# B&R Automation Studio project ACOPOStrak_DATech_Pilot (part 4)

#### Types.typ - Local data types
```iecst
(*estimate assembly power consumption and distribution*)
(*interface structure*)

TYPE
	TrakDesignType : 	STRUCT
		AssemblyRef : REFERENCE TO McAssemblyType; (*assembly reference - ADR(gAssembly_1)*)
		AssemblyName : STRING[32]; (*assembly name - 'gAssembly_1'*)
		EnableCalc : BOOL; (*enable*)
		CmdReset : BOOL; (*command reset peak values*)
		CmdSaveReport : BOOL; (*command save report to file*)
		CmdRecordToolData : BOOL; (*command activate recording of TrakDesign-Tool data*)
		ParaShuttleType : TrakDesignShuttleTypeEnum; (*parameter shuttle type
SA100_50D......8F1SA.100.xxxxxx-1  50mm double sided magnet
SA102_50N......8F1SA.102.xxxxxx-1  50mm single sided magnet
SA201_100D....8F1SA.201.xxxxxx-1  100mm double sided magnet
SA203_100N....8F1SA.203.xxxxxx-1  100mm single sided magnet
SA104_50DS....8F1SA.104.xxxxxx-1  50mm double sided skewed magnet
SA106_50NS....8F1SA.106.xxxxxx-1  50mm single sided skewed magnet
SB308_210N....8F1SB.308.xxxxxx-1  21magnet pole single sided magnet*)
		ParaTempAmbient : REAL; (*parameter ambient air temperature [°C]*)
		ParaMechShuttleIx : UINT; (*parameter mechanical check - use shuttle index*)
		ParaFileDevice : STRING[32]; (*parameter FileDevice*)
		ParaFileNameReport : STRING[32]; (*parameter report file name - file extention .csv mandatory*)
		ParaFileNameToolData : STRING[32]; (*parameter TrakDesign-Tool data file name - file extention .dat mandatory*)
		ParaFileCsvStyle : USINT; (*parameter file csv style
0..english
1..german
2..mathlab*)
		ParaToolDataPrescale : USINT; (*parameter TrakDesign-Tool data prescaler - record TrakDesign-Tool data every x task cycles*)
		Message : STRING[256]; (*message*)
		TimeAsmPowerOn : REAL; (*monitor time elapsed since AsmPowerOn*)
		TimeShuttlesMoving : REAL; (*monitor time shuttles moving - for stabile Avg values process needs to run for >120sec*)
		TimeReset : REAL; (*monitor time elapsed since CmdReset*)
		TimeRecordToolDataActive : REAL; (*monitor time recording of TrakDesign-Tool data active*)
		NumShuttles : UINT; (*monitor number of shuttles present*)
		Carrier : TrakDesignCarrierType;
		Payload : ARRAY[1..8]OF TrakDesignPayloadType;
		Shuttle : ARRAY[1..TRAK_MAX_SHUTTLE]OF TrakDesignShuttleType;
		Segment : ARRAY[1..TRAK_MAX_SEGMENT]OF TrakDesignSegmentType;
		Cable : ARRAY[1..TRAK_MAX_POWER_CABLE]OF TrakDesignCableType;
		Supply : ARRAY[1..TRAK_MAX_POWER_SUPPLY]OF TrakDesignSupplyType;
		MainSupply : TrakDesignMainSupplyType;
		Mech : TrakDesignMechType;
	END_STRUCT;
	TrakDesignCarrierType : 	STRUCT
		ParaMass : LREAL; (*parameter payload carrier mass [kg]*)
		ParaMassCenterX : LREAL; (*parameter payload carrier mass center of gravity offset X [m] (measured from center of shuttle, sign according to the shuttle coordinate system)*)
		ParaMassCenterY : LREAL; (*parameter payload carrier mass center of gravity offset Y [m] (measured from center of shuttle, sign according to the shuttle coordinate system)*)
		ParaMassCenterZ : LREAL; (*parameter payload carrier mass center of gravity offset Z [m] (measured from center of shuttle, sign according to the shuttle coordinate system)*)
		ParaMassInertiaZZ : LREAL; (*parameter payload carrier inertia ZZ [kgm? (with respect to the center of gravity of the carrier - set to 0.0 if unknown)*)
	END_STRUCT;
	TrakDesignPayloadType : 	STRUCT
		ParaName : STRING[32]; (*parameter payload name (free definable name for identification of payload in report and mathlab)*)
		ParaMass : LREAL; (*parameter payload product mass [kg]*)
		ParaMassCenterX : LREAL; (*parameter payload product mass center of gravity offset X [m] (measured from center of shuttle, sign according to the shuttle coordinate system)*)
		ParaMassCenterY : LREAL; (*parameter payload product mass center of gravity offset Y [m] (measured from center of shuttle, sign according to the shuttle coordinate system)*)
		ParaMassCenterZ : LREAL; (*parameter payload product mass center of gravity offset Z [m] (measured from center of shuttle, sign according to the shuttle coordinate system)*)
		ParaMassInertiaZZ : LREAL; (*parameter payload product inertia ZZ [kgm? (with respect to the center of gravity of the payload - set to 0.0 if unknown)*)
		ParaExtFrictionX : LREAL; (*parameter external process friction [N] (sign according to the shuttle movement direction)*)
		ParaExtFrictionVelX : LREAL; (*parameter external process velocity-friction [N/(m/s)] (sign according to the shuttle movement direction)*)
		ParaExtForceX : LREAL; (*parameter external process force X [N] (sign according to the shuttle coordinate system)*)
		ParaExtForceY : LREAL; (*parameter external process force Y [N] (sign according to the shuttle coordinate system)*)
		ParaExtForceZ : LREAL; (*parameter external process force Z [N] (sign according to the shuttle coordinate system)*)
		ParaExtForceAppPointX : LREAL; (*parameter external process force application point offset X [m] (measured from center of shuttle, sign according to the shuttle coordinate system)*)
		ParaExtForceAppPointY : LREAL; (*parameter external process force application point offset Y [m] (measured from center of shuttle, sign according to the shuttle coordinate system)*)
		ParaExtForceAppPointZ : LREAL; (*parameter external process force application point offset Z [m] (measured from center of shuttle, sign according to the shuttle coordinate system)*)
	END_STRUCT;
	TrakDesignShuttleType : 	STRUCT
		ParaPayloadIx : USINT; (*parameter payload index*)
		ParaAutoPayload : USINT; (*parameter autmatic payload selection 0..set PayloadIx explicit / 1..get payload index from ShSelCtrlParSet index*)
		ParaInitialOrientationFlip : INT; (*the initial orientation is different from the one indicated or located.[-]
  1 --> initial orientation is identical with the indicated or located one
 -1 --> initial orientation is different with the indicated or located one *)
		ID : UINT; (*shuttle ID*)
		Vel : LREAL; (*shuttle velocity [m/s]*)
		Acc : LREAL; (*shuttle acceleration [m/s?*)
		Area : USINT; (*shuttle is in area 0..straight / 1..circular / 2..diverter*)
		Force : REAL; (*shuttle thrust force [N]*)
		Current : REAL; (*shuttle current [A]*)
		PowerCalcAct : REAL; (*monitor current shuttle power [W]*)
		PowerCalcAvg : REAL; (*monitor filtered shuttle power [W]*)
		VelStraightPeak : REAL; (*report peak shuttle velocity in straight trak area [m/s]*)
		AccStraightPeak : REAL; (*report peak shuttle acceleration in straight trak area [m/s?*)
		VelCircularPeak : REAL; (*report peak shuttle velocity in circular trak area [m/s]*)
		AccCircularPeak : REAL; (*report peak shuttle acceleration in circular trak area [m/s?*)
		VelDiverterPeak : REAL; (*report peak shuttle velocity in diverter area [m/s]*)
		AccDiverterPeak : REAL; (*report peak shuttle acceleration in diverter area [m/s?*)
		ForcePeak : REAL; (*report peak shuttle thrust Force [N]*)
		CurrentPeak : REAL; (*report peak shuttle current [A]*)
		PowerCalcActPeak : REAL; (*report peak current shuttle power [W]*)
		PowerCalcAvgPeak : REAL; (*report peak filitered shuttle power [W]*)
		CoilDisabled : USINT; (*report reduced force due to temporary disabled stator coil*)
	END_STRUCT;
	TrakDesignSegmentType : 	STRUCT
		ParaName : STRING[32]; (*parameter segment name
name of segment reference variable of type McSegmentType connected to this segment in SystemDesigner*)
		ParaType : TrakDesignSegmentTypeEnum; (*parameter segment type
TYPE_AA
TYPE_AB
TYPE_BA
TYPE_BB*)
		ParaIxCable : USINT; (*parameter segment connected to cable index*)
		ID : UINT; (*segment ID*)
		PowerCalcAct : REAL; (*monitor current segment power [W]*)
		PowerCalcAvg : REAL; (*monitor filtered segment power [W]*)
		PowerCalcActPeak : REAL; (*report peak current segment power [W]*)
		PowerCalcAvgPeak : REAL; (*report peak filtered segment power [W]*)
		PowerCalcLoss : REAL; (*monitor current segment loss [W]*)
		PowerCalcLoad : REAL; (*monitor filtered segment Load [W]*)
		PowerCalcLossPeak : REAL; (*report peak current segment loss [W]*)
		PowerCalcLoadPeak : REAL; (*report peak filtered segment Load [W]*)
		CurrentBalancer : REAL; (*monitor balancer current [A]*)
		CurrentBalancerPeak : REAL; (*report peak balancer current [A]*)
		CoilDisabled : USINT; (*report reduced force due to temporary disabled stator coil*)
	END_STRUCT;
	TrakDesignCableType : 	STRUCT
		ParaLength : REAL; (*parameter cable length [m]*)
		ParaIxSupply : USINT; (*parameter cable connected to PowerSupply index*)
		PowerCalcAct : REAL; (*monitor current cable power [W]*)
		PowerCalcAvg : REAL; (*monitor filtered cable power [W]*)
		PowerCalcActPeak : REAL; (*report peak cable shuttle power [W]*)
		PowerCalcAvgPeak : REAL; (*report peak cable shuttle power [W]*)
		VoltageDropAct : REAL; (*monitor voltage drop [V]*)
		VoltageDropActPeak : REAL; (*report peak voltage drop [V]*)
	END_STRUCT;
	TrakDesignSupplyType : 	STRUCT
		ParaName : STRING[32]; (*parameter supply name
name of supply reference variable of type McAxisType connected to this BC032 in SystemDesigner*)
		ParaType : TrakDesignSupplyTypeEnum; (*parameter supply type
PS080...80PS080X3.10-01         1kW standalone power supply (ACOPOSmicro)
BC032...8B0C0320HW00.B00-1 2kW backplane power supply (ACOPOSmulti)*)
		ParaIxSupplyParallel : USINT; (*Parameter supply is parallel connected to supply index / 0..no parallel connection*)
		PowerCalcAct : REAL; (*monitor current supply power [W]*)
		PowerCalcAvg : REAL; (*monitor filtered supply power [W]*)
		PowerCalcActPeak : REAL; (*report peak current supply power [W]*)
		PowerCalcAvgPeak : REAL; (*report peak filitered supply power [W]*)
		PowerCalcRetPeak : REAL; (*report peak current return power [W]*)
		PowerMeasAct : REAL; (*monitor current supply power [W] (measured via IO)*)
		PowerMeasAvg : REAL; (*monitor filtered supply power [W] (measured via IO)*)
		PowerMeasActPeak : REAL; (*report peak current supply power [W] (measured via IO)*)
		PowerMeasAvgPeak : REAL; (*report peak filitered supply power [W] (measured via IO)*)
		PowerMeasRetPeak : REAL; (*report peak current return power [W] (measured via IO)*)
		IoPS080 : TrakDesignSupplyIoPS080Type;
		IoBC032 : TrakDesignSupplyIoBC032Type;
	END_STRUCT;
	TrakDesignSupplyIoPS080Type : 	STRUCT
		ModuleOk : BOOL; (*PS080 IO*)
		CurrentLimitActive : BOOL; (*PS080 IO*)
		Voltage : SINT; (*PS080 IO [V]*)
		Current : INT; (*PS080 IO [0.1A]*)
		CmdClearError : BOOL; (*PS080 IO*)
		ErrorOutput : BOOL; (*PS080 IO*)
		ErrorOverload : BOOL; (*PS080 IO*)
		ErrorPhaseDetection : BOOL; (*PS080 IO*)
		ErrorOvertemperature : BOOL; (*PS080 IO*)
		ErrorOvervoltage : BOOL; (*PS080 IO*)
		ChopperActive : BOOL; (*PS080 IO*)
		ErrorChopperTemperature : BOOL; (*PS080 IO*)
		ErrorBleederTemperature : BOOL; (*PS080 IO*)
		ErrorOutput24VDC : BOOL; (*PS080 IO*)
	END_STRUCT;
	TrakDesignSupplyIoBC032Type : 	STRUCT
		ModuleOk : BOOL; (*8B0C0320 IO module OK*)
		Iout : REAL; (*8B0C0320 IO Actual Output current [A]*)
		Uout : REAL; (*8B0C0320 IO Actual Output voltage [V]*)
		CrOk : BOOL; (*8B0C0320 IO state charging relais 1..OK*)
		StatusRunMode : USINT; (*8B0C0320 IO Operating mode 0..INIT / 1..READY / 2..ACTIVE / 3..ERROR*)
		ErrorsPacked : UDINT; (*8B0C0320 IO ErrorsPacked - Register ERROR_REG*)
		WarningsPacked : UDINT; (*8B0C0320 IO WarningsPacked - Register WARN_REG*)
	END_STRUCT;
	TrakDesignMainSupplyType : 	STRUCT
		PowerCalcAct : REAL; (*monitor current main supply power [W]*)
		PowerCalcAvg : REAL; (*monitor filtered main supply power [W]*)
		PowerCalcActPeak : REAL; (*report peak current main supply power [W]*)
		PowerCalcAvgPeak : REAL; (*report peak filitered main supply power [W]*)
		PowerCalcRetPeak : REAL; (*report peak current main return power [W]*)
		PowerMeasAct : REAL; (*monitor current main supply power [W] (measured via IO)*)
		PowerMeasAvg : REAL; (*monitor filtered main supply power [W] (measured via IO)*)
		PowerMeasActPeak : REAL; (*report peak current main supply power [W] (measured via IO)*)
		PowerMeasAvgPeak : REAL; (*report peak filitered main supply power [W] (measured via IO)*)
		PowerMeasRetPeak : REAL; (*report peak current main return power [W] (measured via IO)*)
	END_STRUCT;
	TrakDesignMechType : 	STRUCT
		ShuttleIx : UINT;
		ShuttleID : UINT;
		PayloadIx : USINT; (*parameter payload index*)
		ResultThrust : BOOL; (*report thrust force 0..ok / 1..force insufficient*)
		ResultMech : BOOL; (*report mechanical failure 0..ok / 1..shuttle leaving guiding rails*)
		GlobalFrame : McFrameType;
		SectorName : STRING[32];
		SectorPosition : LREAL;
		SectorVelocity : LREAL;
		SectorAcceleration : LREAL;
		SectorOrientation : McDirectionEnum;
		SegmentValid : ARRAY[0..3]OF BOOL;
		SegmentID : ARRAY[0..3]OF UINT;
		SegmentName : ARRAY[0..3]OF STRING[32];
		SegmentTyp : ARRAY[0..3]OF TrakDesignSegmentTypeEnum;
		SegmentLength : ARRAY[0..3]OF LREAL;
		SegmentPosition : ARRAY[0..3]OF LREAL;
		SegmentFieldMode : ARRAY[0..3]OF McAcpTrakFieldModeEnum;
	END_STRUCT;
END_TYPE

(*interface TrakDesign shuttle online interaction*)

TYPE
	TrakDesignOnlineFunctionJobType : 	STRUCT
		LockNew : UDINT;
		Axis : McAxisType;
		ShuttleID : UINT;
		Cmd : USINT;
		PayloadIx : USINT;
		spare : ARRAY[0..3]OF UDINT;
		LockEnd : UDINT;
	END_STRUCT;
END_TYPE

(*TrakDesign-Tool data (diagnosis-data)*)

TYPE
	TrakDesignDiagParaType : 	STRUCT
		VersionDataStruct : UDINT := 2;
		VersionMappMotion : ARRAY[0..9]OF USINT;
		VersionTrakDesignTask : ARRAY[0..9]OF USINT;
		CycleTime : REAL;
		Prescaler : USINT;
		ShuttleType : UINT;
		TempAmbient : REAL;
		PayloadCnt : UINT;
		Carrier : TrakDesignDiagParaCarrierType;
		Payload : ARRAY[1..8]OF TrakDesignDiagParaPayloadType;
		SegmentCnt : UINT;
		Segment : ARRAY[1..TRAK_MAX_SEGMENT]OF TrakDesignDiagParaSegmentType;
		CableCnt : UINT;
		Cable : ARRAY[1..TRAK_MAX_POWER_CABLE]OF TrakDesignDiagParaCableType;
		SupplyCnt : UINT;
		Supply : ARRAY[1..TRAK_MAX_POWER_SUPPLY]OF TrakDesignDiagParaSupplyType;
	END_STRUCT;
	TrakDesignDiagParaCarrierType : 	STRUCT
		Mass : LREAL;
		MassCenterX : LREAL;
		MassCenterY : LREAL;
		MassCenterZ : LREAL;
		MassInertiaZZ : LREAL;
	END_STRUCT;
	TrakDesignDiagParaPayloadType : 	STRUCT
		Name : STRING[32];
		Mass : LREAL;
		MassCenterX : LREAL;
		MassCenterY : LREAL;
		MassCenterZ : LREAL;
		MassInertiaZZ : LREAL;
		ExtFrictionX : LREAL;
		ExtFrictionVelX : LREAL;
		ExtForceX : LREAL;
		ExtForceY : LREAL;
		ExtForceZ : LREAL;
		ExtForceAppPointX : LREAL;
		ExtForceAppPointY : LREAL;
		ExtForceAppPointZ : LREAL;
	END_STRUCT;
	TrakDesignDiagParaSegmentType : 	STRUCT
		Ix : UINT;
		ID : UINT;
		Name : STRING[32];
		Type : TrakDesignSegmentTypeEnum;
		IxCable : UINT;
	END_STRUCT;
	TrakDesignDiagParaCableType : 	STRUCT
		Ix : UINT;
		Length : REAL;
		IxSupply : UINT;
	END_STRUCT;
	TrakDesignDiagParaSupplyType : 	STRUCT
		Ix : UINT;
		Type : TrakDesignSupplyTypeEnum;
		IxSupplyParallel : UINT;
	END_STRUCT;
	TrakDesignDiagType : 	STRUCT
		RecordIndex : UDINT;
		Time : REAL;
		MechShuttleIx : UINT;
		MechResultThrust : BOOL;
		MechResultMech : BOOL;
		AddData : ARRAY[0..4]OF LREAL;
		SegmentCnt : UINT;
		Segment : ARRAY[1..TRAK_MAX_SEGMENT]OF TrakDesignDiagSegmentType;
		ShuttleCnt : UINT;
		Shuttle : ARRAY[1..TRAK_MAX_SHUTTLE]OF TrakDesignDiagShuttleType;
	END_STRUCT;
	TrakDesignDiagSegmentType : 	STRUCT
		CalcPower : REAL;
		CalcLoss : REAL;
	END_STRUCT;
	TrakDesignDiagShuttleType : 	STRUCT
		ID : UINT;
		GlobalFrame : McFrameType;
		SectorVelocity : LREAL;
		SectorAcceleration : LREAL;
		SectorOrientation : McDirectionEnum;
		PayloadIx : UINT;
		GripperCnt : UINT;
		GripperSegValid : ARRAY[0..3]OF BOOL;
		GripperSegIx : ARRAY[0..3]OF UINT;
		GripperSegPosition : ARRAY[0..3]OF LREAL;
		GripperSegFieldMode : ARRAY[0..3]OF McAcpTrakFieldModeEnum;
	END_STRUCT;
END_TYPE

(*supply-data (ServoSoft-import-data)*)

TYPE
	TrakDesignSupplyDataType : 	STRUCT
		Time : LREAL;
		Power : ARRAY[0..TRAK_MAX_POWER_SUPPLY]OF REAL;
	END_STRUCT;
END_TYPE

(*enum*)

TYPE
	TrakDesignShuttleTypeEnum :
		(
		SHUTTLE_UNDEFINED := 0,
		SA100_50D := 100, (*8F1SA.100.xxxxxx-1  50mm double sided magnet*)
		SA102_50N := 102, (*8F1SA.102.xxxxxx-1  50mm single sided magnet*)
		SA201_100D := 201, (*8F1SA.201.xxxxxx-1  100mm double sided magnet*)
		SA203_100N := 203, (*8F1SA.203.xxxxxx-1  100mm single sided magnet*)
		SA104_50DS := 104, (*8F1SA.104.xxxxxx-1  50mm double sided skewed magnet*)
		SA106_50NS := 106, (*8F1SA.106.xxxxxx-1  50mm single sided skewed magnet*)
		SHUTTLE_205 := 205, (*internal*)
		SHUTTLE_207 := 207, (*internal*)
		SB308_210N := 1308, (*8F1SB.308.xxxxxx-1  21magnet pole single sided magnet*)
		SHUTTLE_9100 := 9100, (*internal*)
		SHUTTLE_65535 := 65535 (*internal*)
		);
	TrakDesignSegmentTypeEnum :
		(
		SEGMENT_UNDEFINED := 0,
		TYPE_AA := 1, (*AA Straight segment*)
		TYPE_AB := 2, (*AB Curved segment*)
		TYPE_BA := 3, (*BA Curved segment*)
		TYPE_BB := 4 (*BB Circular arc segment*)
		);
	TrakDesignSupplyTypeEnum :
		(
		SUPPLY_UNDEFINED := 0,
		PS080 := 1, (*80PS080X3.10-01 1kW standalone power supply (ACOPOSmicro)*)
		BC032 := 2 (*8B0C0320HW00.B00-1 2kW backplane power supply (ACOPOSmulti)*)
		);
	TrakDesignStepGetShuttleEnum :
		(
		TRAK_DISABLED := 0,
		TRAK_WAIT,
		TRAK_GET_SHUTTLE_INIT,
		TRAK_GET_SHUTTLE,
		TRAK_GET_SHUTTLE_WAIT,
		TRAK_INIT,
		TRAK_READY,
		TRAK_ERROR
		);
END_TYPE
```

#### Variables.var - Local variables
```iecst
(*task interface structure*)
VAR
	TrakDesign : TrakDesignType;
END_VAR
(*online interface*)
VAR
	OnlineFunctionJob : ARRAY[0..19] OF TrakDesignOnlineFunctionJobType;
	ShuttleIxFound : UDINT := 0;
	ShuttleIxAdd : UDINT := 0;
END_VAR
(*general*)
VAR
	RTInfo_0 : RTInfo;
	TCCycleTime : LREAL;
	i : UDINT;
	k : UINT;
	m : UINT;
	ErrorMessage : USINT := 0;
	VersionMcAcpTrak : MoVerStruc_typ := (0);
	VersionTrakDesignTask : MoVerStruc_typ := (0);
END_VAR
(*get shuttle axis*)
VAR
	MC_BR_AsmReadInfo_AcpTrak_0 : MC_BR_AsmReadInfo_AcpTrak;
	MC_BR_AsmGetShuttle_AcpTrak_0 : MC_BR_AsmGetShuttle_AcpTrak;
	StepGetShuttle : TrakDesignStepGetShuttleEnum;
	CyclesWaitGetShuttle : UINT := TRAK_MAX_SHUTTLE * 5;
	CntWait : UINT;
	CntShuttle : UINT;
	CntShuttleIdentPowerOn : UDINT;
	CntShuttleAddedOnline : UDINT;
	CntShuttleDeletedOnline : UDINT;
	ShuttleAxis : ARRAY[1..TRAK_MAX_SHUTTLE] OF McAxisType;
	AssemblyOrientation : REAL := 0.0;
END_VAR
(*shutte & segment power*)
VAR
	MC_BR_ShReadInfo_AcpTrak_0 : ARRAY[1..TRAK_MAX_SHUTTLE] OF MC_BR_ShReadInfo_AcpTrak;
	MC_BR_ShReadSegmentInfo_0 : ARRAY[1..TRAK_MAX_SHUTTLE] OF MC_BR_ShReadSegmentInfo_AcpTrak;
	MC_BR_ShReadFrame_AcpTrak_0 : ARRAY[1..TRAK_MAX_SHUTTLE] OF MC_BR_ShReadFrame_AcpTrak;
	ShuttleVelEdge : ARRAY[1..TRAK_MAX_SHUTTLE] OF LREAL;
	ShuttleGravity : ARRAY[1..TRAK_MAX_SHUTTLE] OF LREAL;
	SegmentSetValues : ARRAY[0..3] OF McAcpTrakShSegSetValuesType;
	SegmentLength : ARRAY[1..TRAK_MAX_SEGMENT] OF LREAL;
	SegmentNumCoil : ARRAY[1..TRAK_MAX_SEGMENT] OF UINT;
	SegCableResistance : ARRAY[1..TRAK_MAX_SEGMENT] OF LREAL;
	CableResistance : ARRAY[1..TRAK_MAX_POWER_CABLE] OF LREAL;
	FrameXEdge : ARRAY[1..TRAK_MAX_SHUTTLE] OF LREAL;
	FrameYEdge : ARRAY[1..TRAK_MAX_SHUTTLE] OF LREAL;
	FrameZEdge : ARRAY[1..TRAK_MAX_SHUTTLE] OF LREAL;
	FrameXdiff : LREAL := 0.0;
	FrameYdiff : LREAL := 0.0;
	FrameZdiff : LREAL := 0.0;
	FrameVector : LREAL := 0.0;
END_VAR
(*statistics - average power*)
VAR
	FubAvgShuttle : ARRAY[1..TRAK_MAX_SHUTTLE] OF MTBasicsPT1;
	FubAvgSegment : ARRAY[1..TRAK_MAX_SEGMENT] OF MTBasicsPT1;
	FubLoadSegment : ARRAY[1..TRAK_MAX_SEGMENT] OF MTBasicsPT1;
	FubAvgCable : ARRAY[1..TRAK_MAX_POWER_CABLE] OF MTBasicsPT1;
	FubPeakCable : ARRAY[1..TRAK_MAX_POWER_CABLE] OF MTBasicsPT1;
	FubAvgSupply : ARRAY[1..TRAK_MAX_POWER_SUPPLY] OF MTBasicsPT1;
	FubPeakSupply : ARRAY[1..TRAK_MAX_POWER_SUPPLY] OF MTBasicsPT1;
	FubAvgSupplyMeas : ARRAY[1..TRAK_MAX_POWER_SUPPLY] OF MTBasicsPT1;
	FubPeakSupplyMeas : ARRAY[1..TRAK_MAX_POWER_SUPPLY] OF MTBasicsPT1;
	FubAvgMainSupply : MTBasicsPT1;
	FubPeakMainSupply : MTBasicsPT1;
	FubAvgMainSupplyMeas : MTBasicsPT1;
	FubPeakMainSupplyMeas : MTBasicsPT1;
END_VAR
(*Supply error reset*)
VAR
	WaitIoPS080CmdClear : REAL := 0.0;
	StatusGetSupplyAxisRef : UINT := 0;
	LenGetSupplyAxisRef : UDINT := 0;
	SupplyAxisRef : ARRAY[1..TRAK_MAX_POWER_SUPPLY] OF UDINT;
	MC_Reset_0 : ARRAY[1..TRAK_MAX_POWER_SUPPLY] OF MC_Reset;
END_VAR
(*analyze layout*)
VAR
	CheckLayout : BOOL := FALSE;
	LayoutMessageCnt : UINT;
	LayoutMessagePrio : ARRAY[1..TRAK_MAX_SEGMENT] OF USINT;
	LayoutMessage : ARRAY[1..TRAK_MAX_SEGMENT] OF STRING[200];
END_VAR
(*analyze mechanical situation*)
VAR
	MechResultEventCnt : USINT;
	MechResultEventLog : ARRAY[0..19] OF TrakDesignMechType;
END_VAR
(*collect TrakDesign-Tool data (diagnosis-data)*)
VAR CONSTANT
	TRAK_DIAG_BUFFER_SIZE : UDINT := 1000;
END_VAR
VAR
	DiagBufferStatusAlloc : UINT;
	DiagBufferAdr : UDINT;
	DiagBufferCntIn : UDINT;
	DiagBufferCntOut : UDINT;
	CntDiagPrescale : USINT;
	DiagDataPara : TrakDesignDiagParaType;
	DiagData : TrakDesignDiagType;
END_VAR
(*collect Supply data (ServoSoft-import-data)*)
VAR CONSTANT
	TRAK_SUPPLY_BUFFER_SIZE : UDINT := 20000;
END_VAR
VAR
	SupplyBufferStatusAlloc : UINT;
	SupplyBufferAdr : UDINT;
	SupplyBufferCntIn : UDINT;
	SupplyBufferCntStart : UDINT;
	SupplyBufferCntWrite : UDINT;
	SupplyPowerFilter : ARRAY[0..TRAK_MAX_POWER_SUPPLY] OF REAL;
	SupplyData : TrakDesignSupplyDataType;
	SupplyDataTimer : LREAL := 0.0;
	SupplyDataEnable : BOOL := FALSE;
END_VAR
```

- Action.st (not readable text: treated as protected, skipped)

- File.st (not readable text: treated as protected, skipped)

- solveEquSys.st (not readable text: treated as protected, skipped)

#### LocalFunctions.fun
```iecst
{REDUND_ERROR} FUNCTION solveEquSys : BOOL (*solve the linear matrix equation A*x = b*) (*$GROUP=User,$CAT=User,$GROUPICON=User.png,$CATICON=User.png*)
	VAR_INPUT
		A : REFERENCE TO ARRAY[0..35] OF LREAL;
		b : REFERENCE TO ARRAY[0..5] OF LREAL;
		solution : REFERENCE TO ARRAY[0..5] OF LREAL;
	END_VAR
	VAR
		x : ARRAY[0..5] OF LREAL;
		b_A : ARRAY[0..35] OF LREAL;
		i0 : INT;
		j : INT;
		ipiv : ARRAY[0..5] OF INT;
		jy : INT;
		c : INT;
		iy : INT;
		ix : INT;
		smax : LREAL;
		k : INT;
		s : LREAL;
		ijA : INT;
	END_VAR
END_FUNCTION
```

#### LocalTypes.typ - Local data types
```iecst
(*local structures*)

TYPE
	SegCurrType : 	STRUCT
		Coil : ARRAY[1..44]OF SegCurrCoilType;
	END_STRUCT;
	SegCurrCoilType : 	STRUCT
		ShuttleIx : USINT;
		Prio : USINT;
		Current : REAL;
	END_STRUCT;
	DualTrakSegType : 	STRUCT
		Ix : UINT;
		Type : TrakDesignSegmentTypeEnum;
		Len : LREAL;
		Pos : LREAL;
		DistGap : LREAL;
	END_STRUCT;
END_TYPE

(**)
(*enum*)

TYPE
	StepEnum :
		(
		TRAK_COMMAND := 0,
		TRAK_FILE_PREPARE,
		TRAK_FILE_DELETE,
		TRAK_FILE_CREATE,
		TRAK_FILE_OPEN,
		TRAK_PREPARE_HEADER,
		TRAK_PREPARE_DATA,
		TRAK_FILE_BUFFER,
		TRAK_FILE_READ,
		TRAK_FILE_WRITE,
		TRAK_FILE_CLOSE,
		TRAK_FILE_CLOSE_2,
		TRAK_FILE_COPY_HISTORY,
		TRAK_FILE_CLOSE_ERROR,
		TRAK_MESSAGE_DELAY
		);
END_TYPE

(**)
(*datatyp fo the mechanical simulation*)

TYPE
	System_matrix_typ : 	STRUCT
		column1 : ARRAY[0..5]OF LREAL;
		column2 : ARRAY[0..5]OF LREAL;
		column3 : ARRAY[0..5]OF LREAL;
		column4 : ARRAY[0..5]OF LREAL;
		column5 : ARRAY[0..5]OF LREAL;
		column6 : ARRAY[0..5]OF LREAL;
		column7 : ARRAY[0..5]OF LREAL;
	END_STRUCT;
	Solution_typ : 	STRUCT
		xFj_0 : ARRAY[0..5]OF LREAL;
	END_STRUCT;
	Vec_typ : 	STRUCT
		x : LREAL;
		y : LREAL;
		z : LREAL;
	END_STRUCT;
	Frame_orientation_typ : 	STRUCT
		phi : LREAL;
		theta : LREAL;
		psi : LREAL;
	END_STRUCT;
	SegmentSelectionData_typ : 	STRUCT
		SegmentPosition : LREAL;
		SegmentFieldMode : LREAL;
		SegmentLength : LREAL;
		SegmentID : UINT;
		SegmentTyp : TrakDesignSegmentTypeEnum;
	END_STRUCT;
END_TYPE
```

#### LocalVariables.var - Local variables
```iecst
(*shutte & segment power - used in ACTION CalcShuttleSegmentPower*)
VAR
	ParaShuttleType : TrakDesignShuttleTypeEnum := SHUTTLE_UNDEFINED;
	SysData : ARRAY[0..200] OF LREAL;
	ShData : ARRAY[0..200] OF LREAL;
	ShDataShuttleAny : ARRAY[0..200] OF LREAL;
	CntSetValuesValid : USINT;
	FieldModeActive : BOOL;
	ShuttleOnCircularArea : BOOL := FALSE;
	kF0 : LREAL := 0.0;
	kFk : LREAL := 0.0;
	Isq : LREAL;
	Isd : LREAL;
	Ivec : LREAL := 0.0;
	Isa : LREAL := 0.0;
	Isb : LREAL := 0.0;
	rho_off : LREAL := 0.0;
	rho_sm : LREAL := 0.0;
	rho_cos : LREAL := 0.0;
	rho_sin : LREAL := 0.0;
	Is_U : LREAL := 0.0;
	Is_V : LREAL := 0.0;
	Is_W : LREAL := 0.0;
	c : USINT := 0;
	p : DINT := 0;
	ForceShuttleCalc : LREAL := 0.0;
	PowerShuttleCalcKin : LREAL;
	PowerShuttleCalcAct : LREAL;
	IxSegment : UINT;
	LenSegment : LREAL;
	NumCoilSegment : UINT;
	PosSegment : LREAL;
	PosSegFactor : LREAL;
	SupplyPowerCalcAct : ARRAY[1..TRAK_MAX_POWER_SUPPLY] OF LREAL;
	SupplyRailPower : ARRAY[1..TRAK_MAX_POWER_SUPPLY] OF LREAL;
	SupplyRailPowerMeas : ARRAY[1..TRAK_MAX_POWER_SUPPLY] OF LREAL;
	SupplyRailIx : ARRAY[1..TRAK_MAX_POWER_SUPPLY] OF UDINT;
	SupplyRailCnt : ARRAY[1..TRAK_MAX_POWER_SUPPLY] OF INT;
	CoilPrio : USINT := 0;
	CoilCurr : REAL := 0.0;
	CalcSegCurr : BOOL := FALSE;
	SegCurr : ARRAY[1..TRAK_MAX_SEGMENT] OF SegCurrType;
END_VAR
(*layout*)
VAR
	DualTrakSegCnt0 : USINT := 0;
	DualTrakSeg0 : ARRAY[0..1] OF DualTrakSegType := [2((0))];
	DualTrakSegCnt1 : USINT := 0;
	DualTrakSeg1 : ARRAY[0..1] OF DualTrakSegType := [2((0))];
	DualTrakSegGap : ARRAY[0..2] OF DualTrakSegType := [3((0))];
	DualTrakGapPos : LREAL := 0.0;
	DualTrakGapPosMod : LREAL := 0.0;
END_VAR
(*debug*)
VAR
	FubDelayCalcAct : ARRAY[0..TRAK_MAX_POWER_SUPPLY] OF MTBasicsTimeDelay;
	FubDelayMeasAct : ARRAY[0..TRAK_MAX_POWER_SUPPLY] OF MTBasicsTimeDelay;
END_VAR
(*file history*)
VAR
	CreateFileHistory : BOOL := FALSE;
	DTStructureGetTime_0 : DTStructureGetTime := (0);
	TimeActStruct : DTStructure := (0);
	TimeActString : STRING[32] := '';
	FileNameReportHistory : STRING[64] := '';
	FileNameToolDataHistory : STRING[64] := '';
	FileNameSupplyDataHistory : STRING[64] := '';
END_VAR
(*save report to file*)
VAR
	ExpertReport : BOOL := FALSE; (*additional display of the physical values in the report file*)
	StepReport : StepEnum;
	WaitReport : REAL := 0.0;
	SaveDataSectionMax : UINT;
	SaveDataSection : UINT;
	SaveDataIxMax : UINT;
	SaveDataIx : UINT;
	CntReportError : UINT := 0;
	CntReportWarning : UINT := 0;
	PowerCalcLoadPeak : LREAL := 0.0;
	SegmentTmax : ARRAY[1..TRAK_MAX_SEGMENT] OF LREAL; (*parameter maximum allowed segment temperature [°C] / 0..use default*)
	SegmentT : LREAL;
	LoadE : ARRAY[0..3] OF DINT := [4(0)];
	LoadT : DINT := 0;
	LoadMax : DINT;
	TempString : STRING[32];
	pFileChar : REFERENCE TO USINT;
	FileDelete_0 : FileDelete;
	FileCreate_0 : FileCreate;
	FileWrite_0 : FileWrite;
	FileClose_0 : FileClose;
	FileCopy_0 : FileCopy;
	ReportFileIdent : UDINT;
	ReportFileOffset : UDINT;
	ReportDataBuffer : STRING[100000];
	ReportDataLen : UDINT;
END_VAR
(*save diag to file*)
VAR
	OnlineCmdRecordToolData : BOOL := FALSE;
	StepDiag : StepEnum;
	WaitDiag : REAL := 0.0;
	pDiagBufferOut : REFERENCE TO TrakDesignDiagType;
	FileDelete_1 : FileDelete;
	FileCreate_1 : FileCreate;
	FileOpen_1 : FileOpen;
	FileRead_1 : FileRead;
	FileWrite_1 : FileWrite;
	FileClose_1 : FileClose;
	FileCopy_1 : FileCopy;
	ScnFileName : STRING[32] := '';
	ScnFileIdent : UDINT;
	ScnFileLen : UDINT;
	ScnFileData : ARRAY[0..199999] OF USINT;
	DiagFileIdent : UDINT;
	DiagFileOffset : UDINT;
	DiagDataBuffer : ARRAY[0..299999] OF USINT;
	DiagDataBufferCopy : UDINT;
	DiagDataLen : UDINT;
	DiagDataShuttleCnt : UINT := 0;
END_VAR
(*save supply data to file*)
VAR
	CmdSaveSupplyData : BOOL := FALSE;
	ParaFileNameSupplyData : STRING[32] := '';
	StepSupplyData : StepEnum;
	pSupplyDataBufferOut : REFERENCE TO TrakDesignSupplyDataType;
	FileDelete_2 : FileDelete;
	FileCreate_2 : FileCreate;
	FileWrite_2 : FileWrite;
	FileClose_2 : FileClose;
	FileCopy_2 : FileCopy;
	SupplyFileIdent : UDINT;
	SupplyFileOffset : UDINT;
	SupplyDataBuffer : ARRAY[0..299999] OF USINT;
	SupplyDataLen : UDINT;
	SupplyDataIx : UINT;
END_VAR
(**)
(*#######################################################*)
(*mechanical simulation*)
(*#######################################################*)
(**)
(*Sorting and selection of the actuated segments*)
VAR
	SegmentDataSelection : ARRAY[0..1] OF SegmentSelectionData_typ;
	tempSegmentData : SegmentSelectionData_typ;
	SegmentDataSelection_old : ARRAY[0..1] OF SegmentSelectionData_typ;
	delta_Seg0Pos : LREAL := 0;
	orientation_cal : INT := 1;
END_VAR
(**)
(*diverter doublecomb*)
VAR
	double_comb_old : BOOL := FALSE;
	double_comb : BOOL := FALSE;
	VZ : INT := 0;
	ac_L : LREAL := 0.0;
	ac_R : LREAL := 0.0;
	fm_L : LREAL := 0.0;
	fm_R : LREAL := 0.0;
	distri_fac : LREAL := 0.0;
END_VAR
(**)
(*control variable*)
VAR
	j : USINT := 0;
	k01 : USINT := 0;
END_VAR
(**)
(*Calculation variables*)
VAR
	at_xsh : LREAL := 0.0;
	an_ysh : LREAL := 0.0;
	v : LREAL := 0.0;
	v_old : LREAL := 0.0;
	frame_orientation : Frame_orientation_typ := (phi:=0.0,theta:=0.0,psi:=0.0);
	frame_orientation_old : Frame_orientation_typ := (phi:=0.0,theta:=0.0,psi:=0.0);
	delta_angle : LREAL := 0.0;
	omega_z : LREAL := 0.0;
	omega_z_old : LREAL := 0.0;
	omegaDOT_z : LREAL := 0.0;
	omegaDOT_z_raw : LREAL := 0.0;
	omegaDOT_z_raw_old : LREAL := 0.0;
END_VAR
(**)
VAR
	spinDotTotal : Vec_typ := (x:=0.0,y:=0.0,z:=0.0);
	momentumDotCGtotal : Vec_typ := (x:=0.0,y:=0.0,z:=0.0);
	aCGtotal : Vec_typ := (x:=0.0,y:=0.0,z:=0.0);
	FRredx : LREAL := 0.0;
	MRredCPS : Vec_typ := (x:=0.0,y:=0.0,z:=0.0);
END_VAR
(**)
(*Shuttle parameter*)
VAR
	rCPS2F12 : Vec_typ := (x:=0.0,y:=0.0,z:=0.0);
	rCPS2F34 : Vec_typ := (x:=0.0,y:=0.0,z:=0.0);
	rCPS2F5 : Vec_typ := (x:=0.0,y:=0.0,z:=0.0);
	rCPS2F6 : Vec_typ := (x:=0.0,y:=0.0,z:=0.0);
	rON2CPS : Vec_typ := (x:=0.0,y:=0.0,z:=0.0);
	rCPS2CGsh : Vec_typ := (x:=0.0,y:=0.0,z:=0.0);
	Ishzz : LREAL := 0.0;
	rHelpMRredCPSy : LREAL := 0.0;
	rHelpMRredCPSz : LREAL := 0.0;
	msh : LREAL := 0.0;
END_VAR
(*Magnetic*)
VAR
	rCPS2FmagR : Vec_typ := (x:=0.0,y:=0.0,z:=0.0);
	rCPS2FmagL : Vec_typ := (x:=0.0,y:=0.0,z:=0.0);
	MmagLz : LREAL := 0.0;
	MmagRz : LREAL := 0.0;
	FmagLz : LREAL := 0.0;
	FmagLy : LREAL := 0.0;
	FmagRz : LREAL := 0.0;
	FmagRy : LREAL := 0.0;
	Fshear : LREAL := 0.0;
	Fattraction : LREAL := 0.0;
	FmaxProp : LREAL := 0.0;
END_VAR
(**)
(*Inertia parameter total system*)
VAR
	mtotal : LREAL := 0.0;
	rCPS2CGtotal : Vec_typ := (x:=0.0,y:=0.0,z:=0.0);
	rCGcarrier2CGtotal : Vec_typ := (x:=0.0,y:=0.0,z:=0.0);
	rCGload2CGtotal : Vec_typ := (x:=0.0,y:=0.0,z:=0.0);
	rCGsh2CGtotal : Vec_typ := (x:=0.0,y:=0.0,z:=0.0);
	IxzTotal : LREAL := 0.0;
	IyzTotal : LREAL := 0.0;
	IzzTotal : LREAL := 0.0;
	Fgtotal : Vec_typ := (x:=0.0,y:=0.0,z:=0.0);
END_VAR
(**)
(*Matrices and solution vectors*)
VAR
	brhs : ARRAY[0..5] OF LREAL := [6(0.0)];
	A : System_matrix_typ := (0);
	Solutions6extremeCases : ARRAY[1..6] OF Solution_typ := [6((0))];
	Atemp : ARRAY[0..35] OF LREAL := [36(0.0)];
END_VAR
(**)
(*analyse*)
VAR
	vaild_solution : ARRAY[0..5] OF INT := [6(0)];
	insufficient_mech_power_solution : BOOL := FALSE;
	flyoff : BOOL := FALSE;
	MechThrustFilterCnt : USINT;
	MechResultFilterCnt : USINT;
END_VAR
```

### Program Logical/Source/Utility/srvAudit (IEC)

#### Main.st - Init, cyclic, exit code
```iecst
PROGRAM _INIT
	fbAudit.MpLink := ADR(gAuditTrak);
	fbAudit.Enable := TRUE;
	fbAudit.DeviceName := ADR('Log');

END_PROGRAM

PROGRAM _CYCLIC
	fbAudit();

	IF (fbAudit.Export) AND (fbAudit.CommandDone) THEN
		fbAudit.Export := FALSE;
	END_IF
END_PROGRAM

PROGRAM _EXIT
	fbAudit(Enable := FALSE);

END_PROGRAM
```

#### Variables.var - Local variables
```iecst
VAR
	fbAudit : MpAuditTrail;
END_VAR
```

### ProcessControl.var
```iecst
VAR
	StStage : ARRAY[0..18] OF MyTrakSlotType;
END_VAR
(**)
VAR CONSTANT
	COUNT_OF_SLOT : USINT := 1;
END_VAR
(**)
VAR CONSTANT
	SLOT_COUNT_OF_STAGE1 : USINT := 1;
	SLOT_COUNT_OF_STAGE2 : USINT := 1;
	SLOT_COUNT_OF_STAGE3 : USINT := 1;
	LAST_IDX_OF_STAGE1 : USINT := SLOT_COUNT_OF_STAGE1-1;
	LAST_IDX_OF_STAGE2 : USINT := SLOT_COUNT_OF_STAGE2-1;
	LAST_IDX_OF_STAGE3 : USINT := SLOT_COUNT_OF_STAGE3-1;
END_VAR
(**)
VAR CONSTANT
	LENGTH_OF_CURVE : LREAL := 0.450642056;
	LENGTH_OF_STRAIGHT : LREAL := 0.660000000;
	LENGTH_OF_ARC : LREAL := 0.240000000;
END_VAR
(**)
VAR CONSTANT
	LAST_IDX_OF_STAGE5 : USINT := SLOT_COUNT_OF_STAGE1-1;
	LAST_IDX_OF_STAGE6 : USINT := SLOT_COUNT_OF_STAGE1-1;
	LAST_IDX_OF_STAGE7 : USINT := SLOT_COUNT_OF_STAGE1-1;
END_VAR
(*Position of process point*)
VAR CONSTANT
	POS_STAGE1 : LREAL := 0.1785; (*Can supply*)
	POS_STAGE1_MAX : LREAL := POS_STAGE1 + 0.05; (*Sector Curve 1*)
	POS_STAGE1_MIN : LREAL := POS_STAGE1 - 0.05;
END_VAR
(**)
VAR CONSTANT
	POS_STAGE2 : LREAL := 0.1268; (*TC insert*)
	POS_STAGE2_MAX : LREAL := POS_STAGE2 + 0.05; (*Sector 2*)
	POS_STAGE2_MIN : LREAL := POS_STAGE2 - 0.05;
END_VAR
(**)
VAR CONSTANT
	POS_STAGE3 : LREAL := 0.431; (*TC push*)
	POS_STAGE3_MAX : LREAL := POS_STAGE3 + 0.05; (*Sector 2*)
	POS_STAGE3_MIN : LREAL := POS_STAGE3 - 0.05;
END_VAR
(**)
VAR CONSTANT
	POS_STAGE4 : LREAL := 0.664; (*TC vision*)
	POS_STAGE4_MAX : LREAL := POS_STAGE4 + 0.05; (*Sector 2*)
	POS_STAGE4_MIN : LREAL := POS_STAGE4 - 0.05;
END_VAR
(**)
VAR CONSTANT
	POS_STAGE5 : LREAL := 0.8865; (*TC NG re-insert*)
	POS_STAGE5_MAX : LREAL := POS_STAGE5 + 0.05; (*Sector 2*)
	POS_STAGE5_MIN : LREAL := POS_STAGE5 - 0.05;
END_VAR
(**)
VAR CONSTANT
	POS_STAGE6 : LREAL := 0.985; (*BCR vision*)
	POS_STAGE6_MAX : LREAL := POS_STAGE6 + 0.05; (*Sector 2*)
	POS_STAGE6_MIN : LREAL := POS_STAGE6 - 0.05;
END_VAR
(**)
VAR CONSTANT
	POS_STAGE7 : LREAL := 2.18; (*CCR 1*)
	POS_STAGE7_MAX : LREAL := POS_STAGE7 + 0.05; (*Sector 2*)
	POS_STAGE7_MIN : LREAL := POS_STAGE7 - 0.05;
END_VAR
(**)
VAR CONSTANT
	POS_STAGE8 : LREAL := 2.6265; (*CCR 1 vision*)
	POS_STAGE8_MAX : LREAL := POS_STAGE8 + 0.05; (*Sector 2*)
	POS_STAGE8_MIN : LREAL := POS_STAGE8 - 0.05;
END_VAR
(**)
VAR CONSTANT
	POS_STAGE9 : LREAL := 3.1; (*CCR 2*)
	POS_STAGE9_MAX : LREAL := POS_STAGE9 + 0.05; (*Sector 2*)
	POS_STAGE9_MIN : LREAL := POS_STAGE9 - 0.05;
END_VAR
(**)
VAR CONSTANT
	POS_STAGE10 : LREAL := 0.75; (*Maint*)
	POS_STAGE10_MAX : LREAL := POS_STAGE10 + 0.05; (*Sector 3*)
	POS_STAGE10_MIN : LREAL := POS_STAGE10 - 0.05;
END_VAR
(**)
VAR CONSTANT
	POS_STAGE11 : LREAL := 1.052; (*CCR 2 vision*)
	POS_STAGE11_MAX : LREAL := POS_STAGE11 + 0.05; (*Sector Curve 3*)
	POS_STAGE11_MIN : LREAL := POS_STAGE11 - 0.05;
END_VAR
(**)
VAR CONSTANT
	POS_STAGE12 : LREAL := 0.3295; (*CCR 3*)
	POS_STAGE12_MAX : LREAL := POS_STAGE12 + 0.05; (*Sector 4*)
	POS_STAGE12_MIN : LREAL := POS_STAGE12 - 0.05;
END_VAR
(**)
VAR CONSTANT
	POS_STAGE13 : LREAL := 0.9897; (*CCR 3 vision*)
	POS_STAGE13_MAX : LREAL := POS_STAGE13 + 0.05; (*Sector 4*)
	POS_STAGE13_MIN : LREAL := POS_STAGE13 - 0.05;
END_VAR
(**)
VAR CONSTANT
	POS_STAGE14 : LREAL := 1.9586; (*CSZ*)
	POS_STAGE14_MAX : LREAL := POS_STAGE14 + 0.05; (*Sector 4*)
	POS_STAGE14_MIN : LREAL := POS_STAGE14 - 0.05;
END_VAR
(**)
VAR CONSTANT
	POS_STAGE15 : LREAL := 2.7; (*3D vision done position*)
	POS_STAGE15_MAX : LREAL := POS_STAGE15 + 0.05; (*Sector 4*)
	POS_STAGE15_MIN : LREAL := POS_STAGE15 - 0.05;
END_VAR
(**)
VAR CONSTANT
	POS_STAGE16 : LREAL := 2.812; (*Diameter inspection*)
	POS_STAGE16_MAX : LREAL := POS_STAGE16 + 0.05; (*Sector 4*)
	POS_STAGE16_MIN : LREAL := POS_STAGE16 - 0.05;
END_VAR
(**)
VAR CONSTANT
	POS_STAGE17 : LREAL := 0.061; (*NG out*)
	POS_STAGE17_MAX : LREAL := POS_STAGE17 + 0.05; (*Sector Curve 4*)
	POS_STAGE17_MIN : LREAL := POS_STAGE17 - 0.05;
END_VAR
(**)
VAR CONSTANT
	POS_STAGE18 : LREAL := 0.8669; (*Unloading*)
	POS_STAGE18_MAX : LREAL := POS_STAGE18 + 0.05; (*Sector Curve 4*)
	POS_STAGE18_MIN : LREAL := POS_STAGE18 - 0.05;
END_VAR
(**)
VAR CONSTANT
	POS_STAGE19 : LREAL := 0.55; (*Clean*)
	POS_STAGE19_MAX : LREAL := POS_STAGE19 + 0.05; (*Sector 1*)
	POS_STAGE19_MIN : LREAL := POS_STAGE19 - 0.05;
END_VAR
(**)
VAR CONSTANT
	POS_VISION : LREAL := 7.57;
END_VAR
```

### ProcessControl.typ
```iecst
TYPE
	Com_Equip_Side_type : 	STRUCT
		Interlock : BOOL;
		Ready : BOOL;
		Done : BOOL;
		Data : ARRAY[0..8]OF UINT; (*UINT[0..8]*)
		Data2 : ARRAY[0..19]OF UINT;
	END_STRUCT;
	Com_Trak_Side_type : 	STRUCT
		ShuttleArrived : BOOL;
		Data : ARRAY[0..8]OF UINT;
		ShuttleID : REFERENCE TO STRING[11];
		Data2 : ARRAY[0..19]OF UINT;
	END_STRUCT;
	Interface_Process : 	STRUCT
		Equipment : Com_Equip_Side_type;
		Trak : Com_Trak_Side_type;
	END_STRUCT;
	Interface_Process_1Sh : 	STRUCT
		Equipment : Com_Equip_Side_1Sh_type;
		Trak : Com_Trak_Side_1Sh_type;
	END_STRUCT;
	Com_Equip_Side_1Sh_type : 	STRUCT
		Interlock : BOOL;
		Ready : BOOL;
		Busy : BOOL; (*Delete After Modify All*)
		Done : BOOL;
		Data : ARRAY[0..8]OF UINT; (*UINT[0..8]*)
		Data2 : ARRAY[0..19]OF UINT;
	END_STRUCT;
	Com_Trak_Side_1Sh_type : 	STRUCT
		ProcessReq : BOOL; (*Delete After Modify All*)
		ProcessDone : BOOL; (*Delete After Modify All*)
		ShuttleArrived : BOOL;
		Data : ARRAY[0..8]OF UINT; (*UINT[0..8]*)
		Data2 : ARRAY[0..19]OF UINT;
		ShuttleID : REFERENCE TO STRING[11];
	END_STRUCT;
END_TYPE
```

### Program Logical/Source/AsmControl/CtrlAsm (IEC)

#### Main.st - Init, cyclic, exit code
```iecst
PROGRAM _INIT
	fbAsmPowerOff.Assembly 		:= ADR(gAsmMain);
	fbAsmPowerOn.Assembly 		:= ADR(gAsmMain);
	fbAsmReset.Assembly 		:= ADR(gAsmMain);
	fbAsmStop.Assembly 			:= ADR(gAsmMain);
	fbAsmReadStatus.Assembly 	:= ADR(gAsmMain);
	fbAsmReadErrorInfo.Assembly := ADR(gAsmMain);
	fbAsmReadInfo.Assembly 		:= ADR(gAsmMain);
	fbAsmGetShuttle.Assembly	:= ADR(gAsmMain);
END_PROGRAM

PROGRAM _CYCLIC

	// PC running hours
	RunningTime	:= DINT_TO_UDINT(OperatingHours);
	SystemTime	:= UDINT_TO_UINT(RunningTime / 1000000);

	IF gLocal THEN
		cmdPowerOn(CLK := gCmd.PowerOn);
		cmdPowerOff(CLK := gCmd.PowerOff);
		cmdInit(CLK := gCmd.Initialize);
		cmdEMS(CLK := gCmd.EMS);
		cmdStart(CLK := gCmd.Start);
		cmdStop(CLK := gCmd.Stop);
		cmdReset(CLK := gCmd.Reset);
		cmdClean(CLK := gCmd.Clean);
	ELSE
		cmdPowerOn(CLK := gCmdRemote.PowerOn);
		cmdPowerOff(CLK := gCmdRemote.PowerOff);
		cmdInit(CLK := gCmdRemote.Initialize);
		cmdEMS(CLK := gCmdRemote.EMS);
		cmdStart(CLK := gCmdRemote.Start);
		cmdStop(CLK := gCmdRemote.Stop);
		cmdReset(CLK := gCmdRemote.Reset);
		cmdClean(CLK := gCmdRemote.Clean);
	END_IF

	fbAsmReadStatus(Enable := TRUE);

	// Power on/off signal
	IF fbAsmReadInfo.AssemblyInfo.PowerOn THEN
		gStsPowerOn		:= TRUE;
		gStsPowerOff	:= FALSE;
	ELSIF NOT(fbAsmReadInfo.AssemblyInfo.PowerOn) THEN
		gStsPowerOn		:= FALSE;
		gStsPowerOff	:= TRUE;
	END_IF

	// Reset
	IF gCmdRemote.Reset THEN
		gCmd.Reset	:= TRUE;
	ELSIF NOT(gCmdRemote.Reset) THEN
		gCmd.Reset	:= FALSE;
	END_IF

	// EMS
	IF gCmd.EMS OR gCmdRemote.EMS THEN
		gSts.AsmState	:= E_ASM_EMS;
	END_IF

	IF fbAsmReadStatus.AssemblyErrorStop = TRUE AND
		(gSts.AsmState <> E_ASM_ERRORSTOP AND
		gSts.AsmState <> E_ASM_RESET) THEN
		gSts.AsmState := E_ASM_ERRORSTOP;
	END_IF

	CASE gSts.AsmState OF
		E_ASM_UNKNOWN:

			gStsInitialize	:= FALSE;
			gStsEMS			:= FALSE;
			gStsProcess		:= FALSE;
			gStsStopping	:= FALSE;
			gStsIdle		:= FALSE;
			gStsManual		:= FALSE;
			gStsAsmOn		:= FALSE;
			gStsAsmOff		:= FALSE;
			gStsErrorStop	:= FALSE;

			IF fbAsmReadInfo.AssemblyInfo.ReadyForPowerOn = TRUE THEN
				gSts.AsmState := E_ASM_OFF;
			END_IF

		E_ASM_OFF:

			gStsInitialize	:= FALSE;
			gStsEMS			:= FALSE;
			gStsProcess		:= FALSE;
			gStsStopping	:= FALSE;
			gStsIdle		:= FALSE;
			gStsManual		:= FALSE;
			gStsAsmOn		:= FALSE;
			gStsAsmOff		:= TRUE;
			gStsErrorStop	:= FALSE;

			IF fbAsmReadInfo.AssemblyInfo.ReadyForPowerOn = FALSE THEN
				gSts.AsmState := E_ASM_UNKNOWN;
			ELSIF cmdPowerOn.Q = TRUE THEN
				gSts.AsmState := E_ASM_POWER_ON;
			END_IF

		E_ASM_ON:

			gStsInitialize	:= FALSE;
			gStsEMS			:= FALSE;
			gStsProcess		:= FALSE;
			gStsStopping	:= FALSE;
			gStsIdle		:= FALSE;
			gStsManual		:= FALSE;
			gStsAsmOn		:= TRUE;
			gStsAsmOff		:= FALSE;
			gStsErrorStop	:= FALSE;

			IF cmdPowerOff.Q = TRUE THEN
				gSts.AsmState := E_ASM_POWER_OFF;
			ELSIF cmdInit.Q = TRUE THEN
				gSts.AsmState := E_ASM_INITIALIZATION;
			ELSIF NOT(fbAsmReadInfo.AssemblyInfo.PowerOn) THEN
				gSts.AsmState := E_ASM_OFF;
			ELSIF cmdClean.Q THEN
				gSts.AsmState := E_ASM_CLEAN;
			END_IF

		E_ASM_ERRORSTOP:

			gStsInitialize	:= FALSE;
			gStsEMS			:= FALSE;
			gStsProcess		:= FALSE;
			gStsStopping	:= FALSE;
			gStsIdle		:= FALSE;
			gStsManual		:= FALSE;
			gStsAsmOn		:= FALSE;
			gStsAsmOff		:= FALSE;
			gStsErrorStop	:= TRUE;

			IF cmdPowerOff.Q = TRUE THEN
				gSts.AsmState := E_ASM_POWER_OFF;
			ELSIF cmdReset.Q = TRUE THEN
				gSts.AsmState := E_ASM_RESET;
			END_IF

		E_ASM_IDLE:

			gStsInitialize	:= FALSE;
			gStsEMS			:= FALSE;
			gStsProcess		:= FALSE;
			gStsStopping	:= FALSE;
			gStsIdle		:= TRUE;
			gStsManual		:= FALSE;
			gStsAsmOn		:= FALSE;
			gStsAsmOff		:= FALSE;
			gStsErrorStop	:= FALSE;

			IF gManual = TRUE THEN
				gSts.AsmState := E_ASM_MANUAL;
			ELSIF cmdEMS.Q = TRUE THEN
				gSts.AsmState := E_ASM_EMS;
			ELSIF cmdStart.Q = TRUE THEN
				gSts.AsmState := E_ASM_PROCESS;
			ELSIF cmdPowerOff.Q = TRUE THEN
				gSts.AsmState := E_ASM_POWER_OFF;
			END_IF

		E_ASM_MANUAL:

			gStsInitialize	:= FALSE;
			gStsEMS			:= FALSE;
			gStsProcess		:= FALSE;
			gStsStopping	:= FALSE;
			gStsIdle		:= FALSE;
			gStsManual		:= TRUE;
			gStsAsmOn		:= FALSE;
			gStsAsmOff		:= FALSE;
			gStsErrorStop	:= FALSE;

			IF gManual = FALSE THEN
				gSts.AsmState := E_ASM_EMS;
			END_IF

		E_ASM_PROCESS:

			gStsInitialize	:= FALSE;
			gStsEMS			:= FALSE;
			gStsProcess		:= TRUE;
			gStsStopping	:= FALSE;
			gStsIdle		:= FALSE;
			gStsManual		:= FALSE;
			gStsAsmOn		:= FALSE;
			gStsAsmOff		:= FALSE;
			gStsErrorStop	:= FALSE;

			IF cmdEMS.Q = TRUE THEN
				gSts.AsmState := E_ASM_EMS;
			ELSIF cmdStop.Q = TRUE THEN
				gSts.AsmState := E_ASM_STOPPING;
			END_IF

		E_ASM_POWER_ON:

			gStsInitialize	:= FALSE;
			gStsEMS			:= FALSE;
			gStsProcess		:= FALSE;
			gStsStopping	:= FALSE;
			gStsIdle		:= FALSE;
			gStsManual		:= FALSE;
			gStsAsmOn		:= FALSE;
			gStsAsmOff		:= FALSE;
			gStsErrorStop	:= FALSE;

			actPowerOn;

		E_ASM_POWER_OFF:

			gStsInitialize	:= FALSE;
			gStsEMS			:= FALSE;
			gStsProcess		:= FALSE;
			gStsStopping	:= FALSE;
			gStsIdle		:= FALSE;
			gStsManual		:= FALSE;
			gStsAsmOn		:= FALSE;
			gStsAsmOff		:= FALSE;
			gStsErrorStop	:= FALSE;

			actPowerOff;

		E_ASM_RESET:

			gStsInitialize	:= FALSE;
			gStsEMS			:= FALSE;
			gStsProcess		:= FALSE;
			gStsStopping	:= FALSE;
			gStsIdle		:= FALSE;
			gStsManual		:= FALSE;
			gStsAsmOn		:= FALSE;
			gStsAsmOff		:= FALSE;
			gStsErrorStop	:= FALSE;

			actErrorReset;

		E_ASM_EMS:

			gStsInitialize	:= FALSE;
			gStsEMS			:= TRUE;
			gStsProcess		:= FALSE;
			gStsStopping	:= FALSE;
			gStsIdle		:= FALSE;
			gStsManual		:= FALSE;
			gStsAsmOn		:= FALSE;
			gStsAsmOff		:= FALSE;
			gStsErrorStop	:= FALSE;

			actEMS;

		E_ASM_INITIALIZATION:

			gStsInitialize	:= TRUE;
			gStsEMS			:= FALSE;
			gStsProcess		:= FALSE;
			gStsStopping	:= FALSE;
			gStsIdle		:= FALSE;
			gStsManual		:= FALSE;
			gStsAsmOn		:= FALSE;
			gStsAsmOff		:= FALSE;
			gStsErrorStop	:= FALSE;
			//Customeizing

		E_ASM_RECOVERY:
			//Customeizing

		E_ASM_STOPPING:

			gStsInitialize	:= FALSE;
			gStsEMS			:= FALSE;
			gStsProcess		:= FALSE;
			gStsStopping	:= TRUE;
			gStsReset		:= FALSE;
			gStsIdle		:= FALSE;
			gStsManual		:= FALSE;
			gStsAsmOn		:= FALSE;
			gStsAsmOff		:= FALSE;
			gStsErrorStop	:= FALSE;

			IF cmdStart.Q THEN
				gSts.AsmState	:= E_ASM_PROCESS;
			END_IF

		E_ASM_CLEAN:

			gStsInitialize	:= FALSE;
			gStsEMS			:= FALSE;
			gStsProcess		:= FALSE;
			gStsStopping	:= FALSE;
			gStsIdle		:= FALSE;
			gStsManual		:= FALSE;
			gStsAsmOn		:= FALSE;
			gStsAsmOff		:= FALSE;
			gStsErrorStop	:= FALSE;
	END_CASE;

	fbAsmReadStatus(Enable := TRUE);
	fbAsmReadErrorInfo();
	fbAsmReadInfo(Enable := TRUE);

	fbAsmPowerOn();
	fbAsmPowerOff();
	fbAsmReset();
	fbAsmStop();
	fbAsmGetShuttle();
	fbUserData();

	gCmd.PowerOn 	:= FALSE;
	gCmd.PowerOff 	:= FALSE;
	gCmd.Initialize := FALSE;
	gCmd.EMS 		:= FALSE;
	gCmd.Start 		:= FALSE;
	gCmd.Stop 		:= FALSE;
	gCmd.Clean		:= FALSE;

	gCmdRemote.PowerOn 		:= FALSE;
	gCmdRemote.PowerOff 	:= FALSE;
	gCmdRemote.Initialize 	:= FALSE;
	gCmdRemote.EMS 			:= FALSE;
	gCmdRemote.Start 		:= FALSE;
	gCmdRemote.Stop 		:= FALSE;
	gCmdRemote.Reset 		:= FALSE;
	gCmdRemote.Clean		:= FALSE;

END_PROGRAM
```

#### Variables.var - Local variables
```iecst
(**)
VAR
	fbAsmPowerOn : MC_BR_AsmPowerOn_AcpTrak;
	fbAsmPowerOff : MC_BR_AsmPowerOff_AcpTrak;
	fbAsmReset : MC_BR_AsmReset_AcpTrak;
	fbAsmStop : MC_BR_AsmStop_AcpTrak;
	fbAsmGetShuttle : MC_BR_AsmGetShuttle_AcpTrak;
	fbUserData : MC_BR_ShCopyUserData_AcpTrak;
	fbReset : MC_BR_SegReset_AcpTrak;
	fbAsmReadErrorInfo : MC_BR_AsmReadErrorInfo_AcpTrak;
	fbAsmReadInfo : MC_BR_AsmReadInfo_AcpTrak;
	fbAsmReadStatus : MC_BR_AsmReadStatus_AcpTrak;
END_VAR
(**)
VAR
	cmdPowerOn : R_TRIG;
	cmdPowerOff : R_TRIG;
	cmdInit : R_TRIG;
	cmdEMS : R_TRIG;
	cmdStart : R_TRIG;
	cmdStop : R_TRIG;
	cmdReset : R_TRIG;
	cmdTeaching : R_TRIG;
	cmdClean : R_TRIG;
END_VAR
(**)
VAR
	UserData : ShuttleUserData_typ;
END_VAR
(**)
VAR
	ShuttleCount : USINT;
	StrShuttleCount : STRING[80];
END_VAR
(**)
VAR
	gStsPowerOn : BOOL;
	gStsPowerOff : BOOL;
	gStsInitialize : BOOL;
	gStsEMS : BOOL;
	gStsProcess : BOOL;
	gStsStopping : BOOL;
	gStsReset : BOOL;
	gStsIdle : BOOL;
	gStsReady : BOOL;
	gStsManual : BOOL;
	gStsLocal : BOOL;
	gStsAsmOn : BOOL;
	gStsAsmOff : BOOL;
	gStsErrorStop : BOOL;
END_VAR
(**)
VAR
	OperatingHours : DINT;
	RunningTime : UDINT;
	SystemTime : UINT;
END_VAR
```

#### actions.st
```iecst
ACTION actCommandCheck:
	IF gLocal = TRUE THEN
		cmdPowerOn(CLK := gCmd.PowerOn);
		cmdPowerOff(CLK := gCmd.PowerOff);
		cmdInit(CLK := gCmd.Initialize);
		cmdEMS(CLK := gCmd.EMS);
		cmdStart(CLK := gCmd.Start);
		cmdStop(CLK := gCmd.Stop);
	ELSE
		cmdPowerOn(CLK := gCmdRemote.PowerOn);
		cmdPowerOff(CLK := gCmdRemote.PowerOff);
		cmdInit(CLK := gCmdRemote.Initialize);
		cmdEMS(CLK := gCmdRemote.EMS);
		cmdStart(CLK := gCmdRemote.Start);
		cmdStop(CLK := gCmdRemote.Stop);
	END_IF

	cmdReset(CLK := gCmd.Reset OR gCmdRemote.Reset);

	gCmd.PowerOn 			:= FALSE;
	gCmd.PowerOff 			:= FALSE;
	gCmd.Initialize 		:= FALSE;
	gCmd.EMS 				:= FALSE;
	gCmd.Start 				:= FALSE;
	gCmd.Stop 				:= FALSE;
	gCmd.Reset 				:= FALSE;

	gCmdRemote.PowerOn 		:= FALSE;
	gCmdRemote.PowerOff 	:= FALSE;
	gCmdRemote.Initialize 	:= FALSE;
	gCmdRemote.EMS 			:= FALSE;
	gCmdRemote.Start 		:= FALSE;
	gCmdRemote.Stop 		:= FALSE;
	gCmdRemote.Reset 		:= FALSE;
END_ACTION

ACTION actPowerOn:
	IF fbAsmReadStatus.AssemblyDisabled = TRUE AND NOT(fbAsmPowerOn.Error OR NOT(fbAsmPowerOn.ErrorID = 0)) THEN
		fbAsmPowerOn.Execute 		:= TRUE;
		ShuttleCount				:= 0;
	ELSIF fbAsmReadStatus.AssemblyReady = TRUE THEN
		fbAsmPowerOn.Execute 		:= FALSE;

		IF fbAsmGetShuttle.Valid = FALSE THEN
			fbAsmGetShuttle.Enable := TRUE;
		ELSE
			fbAsmGetShuttle.Next 	:= FALSE;

			fbUserData.Axis 		:= ADR(fbAsmGetShuttle.Axis);
			fbUserData.Mode 		:= mcACPTRAK_USERDATA_SET;
			fbUserData.Execute 		:= TRUE;
			fbUserData.DataAddress	:= ADR(UserData);
			fbUserData.DataSize		:= SIZEOF(UserData);

			StrShuttleCount 		:= USINT_TO_STRING(ShuttleCount);

			IF ShuttleCount < 10 THEN
				UserData.SerialNumber		:= 'UNDEFINED0';
				UserData.SerialNumber		:= CONCAT(UserData.SerialNumber, StrShuttleCount);
			ELSIF ShuttleCount < 100 THEN
				UserData.SerialNumber		:= 'UNDEFINED';
				UserData.SerialNumber		:= CONCAT(UserData.SerialNumber, StrShuttleCount);
			END_IF

			IF fbUserData.Done = TRUE THEN
				ShuttleCount 		:= ShuttleCount + 1;
				fbUserData.Execute 	:= FALSE;

				IF fbAsmGetShuttle.RemainingCount = 0 THEN
					fbAsmGetShuttle.Enable 	:= FALSE;
					gSts.AsmState 			:= E_ASM_ON;
				ELSE
					fbAsmGetShuttle.Next 	:= TRUE;
				END_IF
			END_IF
		END_IF
	END_IF

	IF fbAsmPowerOn.Error OR NOT(fbAsmPowerOn.ErrorID = 0) THEN
		fbAsmPowerOn.Execute	:= FALSE;
		gSts.AsmState			:= E_ASM_ERRORSTOP;
	END_IF

END_ACTION

ACTION actPowerOff:
	fbAsmPowerOff.Execute := TRUE;

	IF fbAsmPowerOff.Done = TRUE THEN
		fbAsmPowerOff.Execute := FALSE;
		gSts.AsmState := E_ASM_OFF;
	ELSIF fbAsmPowerOff.Error = TRUE THEN
		fbAsmPowerOff.Execute := FALSE;
		gSts.AsmState := E_ASM_ERRORSTOP;
	END_IF
END_ACTION

ACTION actEMS:
	fbAsmStop.Execute := TRUE;

	IF fbAsmStop.Busy = TRUE THEN
		fbAsmStop.Execute := FALSE;
		gSts.AsmState := E_ASM_ON;
	ELSIF fbAsmStop.Error = TRUE THEN
		fbAsmStop.Execute := FALSE;
	END_IF
END_ACTION

ACTION actErrorReset:
	fbAsmReset.Execute := TRUE;

	IF fbAsmReset.Done = TRUE THEN
		fbAsmReset.Execute := FALSE;
		gSts.AsmState := E_ASM_OFF;
	ELSIF fbAsmReset.Error = TRUE THEN
		fbAsmReset.Execute := FALSE;
		gSts.AsmState := E_ASM_ERRORSTOP;
	END_IF

END_ACTION
```

### Program Logical/Source/AsmControl/CtrAsmInitial (IEC)

#### Variables.var
```iecst
VAR
	initStep : INT;
END_VAR
(**)
VAR
	fbSecGetShuttles : MC_BR_SecGetShuttleSel_AcpTrak;
END_VAR
(**)
VAR
	fbMovelVel : MC_BR_RoutedMoveVel_AcpTrak;
	fbMoveAbs : MC_BR_RoutedMoveAbs_AcpTrak;
END_VAR
(**)
VAR
	bMoveVelActive : BOOL;
END_VAR
(**)
VAR
	fbBarCmd : MC_BR_BarrierCommand_AcpTrak;
	fbBarNG : MC_BR_BarrierCommand_AcpTrak;
	fbBarBufferOut : MC_BR_BarrierCommand_AcpTrak;
END_VAR
(**)
VAR
	fbCheckOutStatus : MC_BR_BarrierReadInfo_AcpTrak;
	fbCheckInStatus : MC_BR_BarrierReadInfo_AcpTrak;
	fbCheckIn : MC_BR_BarrierCommand_AcpTrak;
	fbCheckOut : MC_BR_BarrierCommand_AcpTrak;
	fbCheckInTrg : MC_BR_TrgPointEnable_AcpTrak;
	fbCheckInTrgInfo : MC_BR_TrgPointGetInfo_AcpTrak;
END_VAR
(**)
(**)
VAR
	TotalShuttleCount : DINT;
	preSerialNumber : STRING[11];
	CharCount : UDINT;
	fbUserData : MC_BR_ShCopyUserData_AcpTrak;
	fbTrgIdentSh : MC_BR_TrgPointGetInfo_AcpTrak;
	fbTmr : TON;
	userData : ShuttleUserData_typ;
	i : INT;
END_VAR
```

#### Main.st
```iecst
PROGRAM _INIT

	fbCheckIn.ProcessPoint			:= ADR(ptCheckIn);
	fbCheckInStatus.ProcessPoint 	:= ADR(ptCheckIn);
	fbCheckInTrg.ProcessPoint		:= ADR(ptCheckIn);
	fbCheckInTrgInfo.ProcessPoint	:= ADR(ptCheckIn);

	fbCheckOutStatus.ProcessPoint	:= ADR(ptCheckOut);
	fbCheckOut.ProcessPoint			:= ADR(ptCheckOut);

	IF gParInitialized = FALSE THEN
		gPar.MovementPar.Initialize.Velocity := 1.0;
		gPar.MovementPar.Initialize.RoutedVelocity := 1.0;
		gPar.MovementPar.Initialize.Acceleration := 1.0;
		gPar.MovementPar.Initialize.Deceleration := 1.0;

		gPar.TargetPPM := 40;
		gPar.CountOfGroup := 1;
	END_IF

END_PROGRAM

PROGRAM _CYCLIC

	IF gSts.AsmState <> E_ASM_INITIALIZATION THEN
		initStep 						:= 0;
		TotalShuttleCount				:= 0;

		fbSecGetShuttles.Enable 		:= FALSE;

		fbCheckInTrg.Enable				:= FALSE;
		fbCheckInTrgInfo.Execute		:= FALSE;
		fbCheckIn.Execute				:= FALSE;
		fbCheckInStatus.Enable			:= FALSE;
		fbCheckOut.Execute				:= FALSE;
		fbCheckOutStatus.Enable			:= FALSE;

		fbMoveAbs.Execute				:= FALSE;
		fbMovelVel.Execute 				:= FALSE;
	ELSE
		CASE initStep OF
			0:
				fbCheckInStatus.Enable := TRUE;
				fbCheckIn.Execute := TRUE;
				fbCheckOut.Execute := TRUE;
				BrBuffer.Execute := TRUE;

				fbCheckIn.Command := mcACPTRAK_BARRIER_CLOSE;
				fbCheckOut.Command := mcACPTRAK_BARRIER_OPEN;

				BrBuffer.Command := mcACPTRAK_BARRIER_OPEN;

				IF fbCheckIn.Done = TRUE AND fbCheckOut.Done = TRUE AND fbCheckInStatus.Valid = TRUE AND BrBuffer.Done THEN
					fbCheckIn.Execute 			:= FALSE;
					fbCheckOut.Execute 			:= FALSE;
					BrBuffer.Execute 			:= FALSE;
					initStep 					:= 100;
				END_IF

			100:
				fbSecGetShuttles.Sector 		:= ADR(SectorTrackAll);
				fbSecGetShuttles.Enable 		:= TRUE;
				fbSecGetShuttles.AdvancedParameters.StartPosition := 0.0;
				fbSecGetShuttles.AdvancedParameters.EndPosition := 0.0;

				IF fbSecGetShuttles.Valid = TRUE THEN
					TotalShuttleCount 		:= fbSecGetShuttles.TotalCount;
					initStep 				:= 210;
				END_IF

			210:
				fbSecGetShuttles.Next 			:= FALSE;

				fbMovelVel.Sector				:= ADR(SectorTrackAll);
				fbMovelVel.Axis 				:= ADR(fbSecGetShuttles.Axis);

				fbMovelVel.Position				:= 12.48;
				fbMovelVel.RouteVelocity 		:= gPar.MovementPar.Initialize.RoutedVelocity;
				fbMovelVel.Velocity 			:= gPar.MovementPar.Initialize.Velocity;
				fbMovelVel.Acceleration 		:= gPar.MovementPar.Initialize.Acceleration;
				fbMovelVel.Deceleration 		:= gPar.MovementPar.Initialize.Deceleration;
				fbMovelVel.Execute 				:= TRUE;

				fbMovelVel.AdvancedParameters.StartDirection 		:= mcDIR_POSITIVE;
				fbMovelVel.AdvancedParameters.EndDirection 			:= mcDIR_UNDEFINED;
				fbMovelVel.AdvancedParameters.ShuttleOrientation 	:= mcDIR_UNDEFINED;

				IF bMoveVelActive = FALSE AND fbMovelVel.Active = TRUE THEN
					fbMovelVel.Execute 			:= FALSE;
					initStep 					:= 220;
				END_IF

			220:
				IF fbSecGetShuttles.RemainingCount > 0 THEN
					fbSecGetShuttles.Next 		:= TRUE;
					initStep 					:= 210;
				ELSE
					fbSecGetShuttles.Enable 	:= FALSE;
					initStep 					:= 230;
				END_IF

				(* Go To Bar Code Reading *)
				(* Go To Bar Code Reading *)
				(* Go To Bar Code Reading *)
			230:
				fbCheckInTrg.Enable := TRUE;

				IF fbCheckInTrg.Valid = TRUE THEN
					fbCheckIn.Command							:= mcACPTRAK_BARRIER_ADD_TICKETS;
					fbCheckIn.AdvancedParameters.TicketCount 	:= TotalShuttleCount;
					fbCheckIn.Execute							:= TRUE;

					IF fbCheckIn.Done = TRUE THEN
						fbCheckIn.Execute 		:= FALSE;
						initStep 				:= 240;
					END_IF
				END_IF

			240:
				IF fbCheckInTrg.EventCount > 0 THEN
					initStep 				:= 250;
				END_IF

			250:
				fbCheckInTrgInfo.Execute := TRUE;

				IF fbCheckInTrgInfo.Done = TRUE THEN
					initStep 				:= 260;
				END_IF

			260:
				fbMoveAbs.Sector		:= ADR(SectorTrackAll);
				fbMoveAbs.Axis			:= ADR(fbCheckInTrgInfo.TrgPointInfo.Axis);
				fbMoveAbs.Position		:= 7.57;//(LENGTH_OF_ARC * 1) + (LENGTH_OF_CURVE * 3) + (LENGTH_OF_STRAIGHT * 5) + 0.12;
				fbMoveAbs.Velocity 		:= gPar.MovementPar.Initialize.Velocity;
				fbMoveAbs.Acceleration 	:= gPar.MovementPar.Initialize.Acceleration;
				fbMoveAbs.Deceleration 	:= gPar.MovementPar.Initialize.Deceleration;
				fbMoveAbs.AdvancedParameters.StartDirection 	:= mcDIR_POSITIVE;
				fbMoveAbs.AdvancedParameters.EndDirection 		:= mcDIR_UNDEFINED;
				fbMoveAbs.AdvancedParameters.ShuttleOrientation := mcDIR_UNDEFINED;
				fbMoveAbs.Execute 		:= TRUE;

				IF fbMoveAbs.Done = TRUE THEN
					fbMoveAbs.Execute 	:= FALSE;
					initStep 			:= 270;
				END_IF

				(* Read User Data *)
			270:

				fbUserData.Axis := ADR(fbCheckInTrgInfo.TrgPointInfo.Axis);
				fbUserData.DataSize := SIZEOF(userData);
				fbUserData.DataAddress := ADR(userData);
				fbUserData.Mode := mcACPTRAK_USERDATA_GET;

				fbUserData.Execute := TRUE;

				IF fbUserData.Done = TRUE THEN
					fbUserData.Execute := FALSE;
					gBarCodeReader.Trigger := TRUE;
					initStep := 271;
				END_IF

				(* Read BCR *)
			271:
				//Timer Check
				IF gSim = TRUE THEN
					initStep := 272;
				END_IF

				CharCount := brsstrlen(ADR(gBarCodeReader.SerialNumber));
				fbTmr(IN := TRUE, PT:= T#5s);

				IF preSerialNumber <> gBarCodeReader.SerialNumber THEN
					//ID Check
					IF CharCount = 11 THEN
						brsmemcpy(ADR(userData.SerialNumber), ADR(gBarCodeReader.SerialNumber), 11);
						brsmemset(ADR(userData.Data),0,SIZEOF(userData.Data));
						initStep := 272;
					ELSE
						gBarCodeReader.Trigger := TRUE;
					END_IF

					fbTmr(IN := FALSE);
				ELSIF fbTmr.Q = TRUE THEN
					gBarCodeReader.Trigger := TRUE;
					fbTmr(IN := FALSE);
				END_IF

				(* Write User Data *)
			272:
				fbUserData.Axis := ADR(fbCheckInTrgInfo.TrgPointInfo.Axis);
				fbUserData.DataSize := SIZEOF(userData);
				fbUserData.DataAddress := ADR(userData);
				fbUserData.Mode := mcACPTRAK_USERDATA_SET;

				fbUserData.Execute := TRUE;

				IF fbUserData.Done = TRUE THEN
					fbUserData.Execute := FALSE;
					initStep := 280;
				END_IF

				(* Move to Home *)
			280:
				fbMovelVel.Sector				:= ADR(SectorTrackAll);
				fbMovelVel.Axis 				:= ADR(fbCheckInTrgInfo.TrgPointInfo.Axis);

				fbMovelVel.Position				:= 12.48;
				fbMovelVel.RouteVelocity 		:= gPar.MovementPar.Initialize.RoutedVelocity;
				fbMovelVel.Velocity 			:= gPar.MovementPar.Initialize.Velocity;
				fbMovelVel.Acceleration 		:= gPar.MovementPar.Initialize.Acceleration;
				fbMovelVel.Deceleration 		:= gPar.MovementPar.Initialize.Deceleration;
				fbMovelVel.Execute 				:= TRUE;

				fbMovelVel.AdvancedParameters.StartDirection 		:= mcDIR_POSITIVE;
				fbMovelVel.AdvancedParameters.EndDirection 			:= mcDIR_UNDEFINED;
				fbMovelVel.AdvancedParameters.ShuttleOrientation 	:= mcDIR_UNDEFINED;

				IF bMoveVelActive = FALSE AND fbMovelVel.Active = TRUE THEN
					TotalShuttleCount 			:= TotalShuttleCount - 1;
					fbMovelVel.Execute 			:= FALSE;
					fbCheckInTrgInfo.Execute 	:= FALSE;

					IF TotalShuttleCount > 0 THEN
						initStep 					:= 240;
					ELSE
						initStep 					:= 300;
					END_IF
				END_IF

			300:
				IF fbCheckInStatus.BarrierInfo.RemainingTickets = 0 THEN
					fbCheckInTrg.Enable			:= FALSE;
					initStep 					:= 400;
				END_IF

			400:
				fbSecGetShuttles.Sector 		:= ADR(SectorTrackAll);
				fbSecGetShuttles.Enable 		:= TRUE;
				fbSecGetShuttles.AdvancedParameters.StartPosition 	:= 13.14;//12.48; // Check in point
				fbSecGetShuttles.AdvancedParameters.EndPosition 	:= 0.0;

				IF fbSecGetShuttles.Valid = TRUE AND fbSecGetShuttles.TotalCount = 0 THEN
					fbSecGetShuttles.Enable 		:= FALSE;
					initStep 						:= 1000;
				ELSIF  fbSecGetShuttles.Valid = TRUE AND fbSecGetShuttles.TotalCount > 0 THEN
					fbSecGetShuttles.Enable 		:= FALSE;
				END_IF

			1000:
				fbCheckInStatus.Enable := FALSE;
				fbCheckIn.Execute := TRUE;
				fbCheckOut.Execute := TRUE;
				BrBuffer.Execute := TRUE;

				fbCheckIn.Command := mcACPTRAK_BARRIER_OPEN;
				fbCheckOut.Command := mcACPTRAK_BARRIER_CLOSE;
				BrBuffer.Command := mcACPTRAK_BARRIER_CLOSE;

				IF fbCheckIn.Done = TRUE AND fbCheckOut.Done = TRUE THEN
					fbCheckIn.Execute 			:= FALSE;
					fbCheckOut.Execute 			:= FALSE;
					fbSecGetShuttles.Enable 	:= FALSE;
					gSts.AsmState 				:= E_ASM_IDLE;

					FOR i := 0 TO 18 DO
						StStage[i].Interface	:= E_SLOT_IDLE;
					END_FOR;

					initStep 					:= 0;
				END_IF

				IF BrBuffer.Done THEN
					BrBuffer.Execute := FALSE;
				END_IF
		END_CASE;
	END_IF

	fbSecGetShuttles();

	fbCheckInTrg();
	fbCheckInTrgInfo();
	fbCheckIn();
	fbCheckInStatus();
	fbCheckOut();
	fbCheckOutStatus();
	fbUserData();

	fbMoveAbs();
	bMoveVelActive 	:= fbMovelVel.Active;
	fbMovelVel();

END_PROGRAM

PROGRAM _EXIT
	fbSecGetShuttles.Enable 		:= FALSE;

	fbCheckInTrg.Enable				:= FALSE;
	fbCheckInTrgInfo.Execute		:= FALSE;
	fbCheckIn.Execute				:= FALSE;
	fbCheckInStatus.Enable			:= FALSE;
	fbCheckOut.Execute				:= FALSE;
	fbCheckOutStatus.Enable			:= FALSE;

	fbMoveAbs.Execute				:= FALSE;
	fbMovelVel.Execute 				:= FALSE;

	fbSecGetShuttles();

	fbCheckInTrg();
	fbCheckInTrgInfo();
	fbCheckIn();
	fbCheckInStatus();
	fbCheckOut();
	fbCheckOutStatus();

	fbMoveAbs();
	fbMovelVel();
END_PROGRAM
```

### Program Logical/Source/AsmControl/CtrAsmInitial2 (IEC)

#### Variables.var
```iecst
VAR
	initStep : INT;
END_VAR
(**)
VAR
	fbSecGetShuttles : MC_BR_SecGetShuttleSel_AcpTrak;
END_VAR
(**)
VAR
	fbMovelVel : MC_BR_RoutedMoveVel_AcpTrak;
END_VAR
(**)
VAR
	bMoveVelActive : BOOL;
END_VAR
(**)
VAR
	fbBarCmd : MC_BR_BarrierCommand_AcpTrak;
	fbBarNG : MC_BR_BarrierCommand_AcpTrak;
	fbBarBufferOut : MC_BR_BarrierCommand_AcpTrak;
END_VAR
(**)
VAR
	fbCheckOutStatus : MC_BR_BarrierReadInfo_AcpTrak;
	fbCheckInStatus : MC_BR_BarrierReadInfo_AcpTrak;
	fbCheckIn : MC_BR_BarrierCommand_AcpTrak;
	fbCheckOut : MC_BR_BarrierCommand_AcpTrak;
	fbEndLimit : MC_BR_BarrierCommand_AcpTrak;
END_VAR
(**)
(**)
VAR
	TotalShuttleCount : DINT;
END_VAR
```

#### Main.st
```iecst
PROGRAM _INIT
//	fbBarBufferOut.ProcessPoint	:= ADR(ptHome);
//	fbBarCmd.ProcessPoint		:= ADR(ptBufferIn);
//	fbBarNG.ProcessPoint 		:= ADR(ptLimitNGArea);

	fbCheckIn.ProcessPoint			:= ADR(ptCheckIn);
	fbCheckInStatus.ProcessPoint 	:= ADR(ptCheckIn);

	fbCheckOutStatus.ProcessPoint	:= ADR(ptCheckOut);
	fbCheckOut.ProcessPoint			:= ADR(ptCheckOut);

	IF gParInitialized = FALSE THEN
		gPar.MovementPar.Initialize.Velocity := 1.0;
		gPar.MovementPar.Initialize.RoutedVelocity := 1.0;
		gPar.MovementPar.Initialize.Acceleration := 1.0;
		gPar.MovementPar.Initialize.Deceleration := 1.0;

		gPar.TargetPPM := 40;
		gPar.CountOfGroup := 1;
	END_IF

END_PROGRAM

PROGRAM _CYCLIC
	IF gSts.AsmState <> E_ASM_INITIALIZATION THEN
		initStep 						:= 0;
		TotalShuttleCount				:= 0;
	ELSE
		CASE initStep OF
			0:(* Process Point Setting *)
				fbCheckInStatus.Enable := TRUE;
				fbCheckIn.Execute := TRUE;
				fbCheckOut.Execute := TRUE;
				fbEndLimit.Execute := TRUE;

				fbCheckIn.Command := mcACPTRAK_BARRIER_CLOSE;
				fbCheckOut.Command := mcACPTRAK_BARRIER_OPEN;

				IF fbCheckIn.Done = TRUE AND fbCheckOut.Done = TRUE AND fbCheckInStatus.Valid = TRUE THEN
					fbCheckIn.Execute 			:= FALSE;
					fbCheckOut.Execute 			:= FALSE;
					initStep 					:= 100;
				END_IF

			100:
				fbSecGetShuttles.Sector 		:= ADR(SectorTrackAll);
				fbSecGetShuttles.Enable 		:= TRUE;
				fbSecGetShuttles.AdvancedParameters.StartPosition := 0.0;
				fbSecGetShuttles.AdvancedParameters.EndPosition := 0.0;

				IF fbSecGetShuttles.Valid = TRUE THEN
					fbCheckIn.Command							:= mcACPTRAK_BARRIER_ADD_TICKETS;
					fbCheckIn.AdvancedParameters.TicketCount 	:= fbSecGetShuttles.TotalCount;
					fbCheckIn.Execute							:= TRUE;

					IF fbCheckIn.Done = TRUE THEN
						fbCheckIn.Execute 		:= FALSE;
						initStep 				:= 210;
					END_IF
				END_IF

			210:
				fbSecGetShuttles.Next 			:= FALSE;

				fbMovelVel.Sector				:= ADR(SectorTrackAll);
				fbMovelVel.Axis 				:= ADR(fbSecGetShuttles.Axis);

				fbMovelVel.Position				:= 12.48;
				fbMovelVel.RouteVelocity 		:= gPar.MovementPar.Initialize.RoutedVelocity;
				fbMovelVel.Velocity 			:= gPar.MovementPar.Initialize.Velocity;
				fbMovelVel.Acceleration 		:= gPar.MovementPar.Initialize.Acceleration;
				fbMovelVel.Deceleration 		:= gPar.MovementPar.Initialize.Deceleration;
				fbMovelVel.Execute 				:= TRUE;

				fbMovelVel.AdvancedParameters.StartDirection 		:= mcDIR_POSITIVE;
				fbMovelVel.AdvancedParameters.EndDirection 			:= mcDIR_UNDEFINED;
				fbMovelVel.AdvancedParameters.ShuttleOrientation 	:= mcDIR_UNDEFINED;

				IF bMoveVelActive = FALSE AND fbMovelVel.Active = TRUE THEN
					fbMovelVel.Execute 			:= FALSE;
					initStep 					:= 220;
				END_IF

			220:
				IF fbSecGetShuttles.RemainingCount > 0 THEN
					fbSecGetShuttles.Next 		:= TRUE;
					initStep 					:= 210;
				ELSE
					fbSecGetShuttles.Enable 	:= FALSE;
					initStep 					:= 300;
				END_IF

			300:
				IF fbCheckInStatus.BarrierInfo.RemainingTickets = 0 THEN
					initStep 					:= 400;
				END_IF

			400:
				fbSecGetShuttles.Sector 		:= ADR(SectorTrackAll);
				fbSecGetShuttles.Enable 		:= TRUE;
				fbSecGetShuttles.AdvancedParameters.StartPosition 	:= 13.14;//12.48; // Check in point
				fbSecGetShuttles.AdvancedParameters.EndPosition 	:= 0.0;

				IF fbSecGetShuttles.Valid = TRUE AND fbSecGetShuttles.TotalCount = 0 THEN
					fbSecGetShuttles.Enable 		:= FALSE;
					initStep 						:= 1000;
				ELSIF  fbSecGetShuttles.Valid = TRUE AND fbSecGetShuttles.TotalCount > 0 THEN
					fbSecGetShuttles.Enable 		:= FALSE;
				END_IF

			1000:
				fbCheckInStatus.Enable := FALSE;
				fbCheckIn.Execute := TRUE;
				fbCheckOut.Execute := TRUE;

				fbCheckIn.Command := mcACPTRAK_BARRIER_OPEN;
				fbCheckOut.Command := mcACPTRAK_BARRIER_CLOSE;

				IF fbCheckIn.Done = TRUE AND fbCheckOut.Done = TRUE THEN
					fbCheckIn.Execute 			:= FALSE;
					fbCheckOut.Execute 			:= FALSE;
					fbSecGetShuttles.Enable 	:= FALSE;
					gSts.AsmState 				:= E_ASM_IDLE;
					initStep 					:= 0;
				END_IF
		END_CASE;
	END_IF

	fbCheckIn();
	fbCheckInStatus();
	fbCheckOut();
	fbCheckOutStatus();

	fbSecGetShuttles();

	bMoveVelActive 	:= fbMovelVel.Active;

	fbMovelVel();

	//	//SecOut 		-> Start Point of SecIn
	//	//SecIn 		-> Start Point of SecIn
	//	//Sector Main 	-> Start Point of SecMain
	//	//SectorIn		-> Start Point of SecMain
	//	//Bar Code Checking
	//
	//	CASE initStep OF
	//		0:
	//			IF gSts.AsmState = E_ASM_INITIALIZATION THEN
	//				initStep 					:= 100;
	//			END_IF
	//
	//		100: (* Barrier Status Setting *)
	//			fbBarBufferOut.Command			:= mcACPTRAK_BARRIER_OPEN;
	//			fbBarBufferOut.Execute 			:= TRUE;
	//
	//			fbBarCmd.Command 				:= mcACPTRAK_BARRIER_CLOSE;
	//			fbBarCmd.Execute 				:= TRUE;
	//
	//
	//
	//			IF fbBarCmd.Done = TRUE AND fbBarBufferOut.Done = TRUE THEN
	//				fbBarBufferOut.Execute 		:= FALSE;
	//				fbBarCmd.Execute 			:= FALSE;
	//				initStep 					:= 101;
	//			END_IF
	//
	//		101:
	//			fbBarNG.Command 				:= mcACPTRAK_BARRIER_CLOSE;
	//			fbBarNG.Execute 				:= TRUE;
	//
	//			IF fbBarNG.Done = TRUE THEN
	//				fbBarNG.Execute 			:= FALSE;
	//				initStep 					:= 110;
	//			END_IF
	//
	//			////////////////////////////////////////////////////////////////////////////////
	//		110:
	//			fbSecGetShuttles.Sector := ADR(SecOut);
	//			fbSecGetShuttles.Enable := TRUE;
	//			fbSecGetShuttles.AdvancedParameters.StartPosition := 0.0;
	//			fbSecGetShuttles.AdvancedParameters.EndPosition := 0.0;
	//
	//			IF fbSecGetShuttles.Valid = TRUE THEN
	//				IF fbSecGetShuttles.TotalCount > 0 THEN
	//					initStep 					:= 111;
	//				ELSE
	//					fbSecGetShuttles.Enable 	:= FALSE;
	//					initStep 					:= 120;
	//				END_IF
	//			END_IF
	//
	//		111:
	//			fbSecGetShuttles.Next 			:= FALSE;
	//
	//			fbMovelVel.Sector				:= ADR(SecIn);
	//			fbMovelVel.Axis 				:= ADR(fbSecGetShuttles.Axis);
	//
	//			fbMovelVel.RouteVelocity 		:= gPar.MovementPar.Initialize.RoutedVelocity;
	//			fbMovelVel.Velocity 			:= gPar.MovementPar.Initialize.Velocity;
	//			fbMovelVel.Acceleration 		:= gPar.MovementPar.Initialize.Acceleration;
	//			fbMovelVel.Deceleration 		:= gPar.MovementPar.Initialize.Deceleration;
	//			fbMovelVel.Execute 				:= TRUE;
	//
	//			fbMovelVel.AdvancedParameters.StartDirection 		:= mcDIR_NEGATIVE;
	//			fbMovelVel.AdvancedParameters.EndDirection 			:= mcDIR_UNDEFINED;
	//			fbMovelVel.AdvancedParameters.ShuttleOrientation 	:= mcDIR_UNDEFINED;
	//
	//			IF bMoveVelActive = FALSE AND fbMovelVel.Active = TRUE THEN
	//				fbMovelVel.Execute 			:= FALSE;
	//				initStep 					:= 112;
	//			END_IF
	//
	//		112:
	//			IF fbSecGetShuttles.RemainingCount > 0 THEN
	//				fbSecGetShuttles.Next 		:= TRUE;
	//				initStep 					:= 111;
	//			ELSE
	//				fbSecGetShuttles.Enable 	:= FALSE;
	//				initStep 					:= 120;
	//			END_IF
	//			////////////////////////////////////////////////////////////////////////////////
	//		120:
	//			fbSecGetShuttles.Sector := ADR(SecIn);
	//			fbSecGetShuttles.Enable := TRUE;
	//			fbSecGetShuttles.AdvancedParameters.StartPosition := 0.0;
	//			fbSecGetShuttles.AdvancedParameters.EndPosition := 2.55;
	//
	//			IF fbSecGetShuttles.Valid = TRUE THEN
	//				IF fbSecGetShuttles.TotalCount > 0 THEN
	//					initStep 					:= 121;
	//				ELSE
	//					fbSecGetShuttles.Enable 	:= FALSE;
	//					initStep 					:= 130;
	//				END_IF
	//			END_IF
	//
	//		121:
	//			fbSecGetShuttles.Next 			:= FALSE;
	//
	//			fbMovelVel.Sector				:= ADR(SecIn);
	//			fbMovelVel.Axis 				:= ADR(fbSecGetShuttles.Axis);
	//
	//			fbMovelVel.RouteVelocity 		:= gPar.MovementPar.Initialize.RoutedVelocity;
	//			fbMovelVel.Velocity 			:= gPar.MovementPar.Initialize.Velocity;
	//			fbMovelVel.Acceleration 		:= gPar.MovementPar.Initialize.Acceleration;
	//			fbMovelVel.Deceleration 		:= gPar.MovementPar.Initialize.Deceleration;
	//			fbMovelVel.Execute 				:= TRUE;
	//
	//			fbMovelVel.AdvancedParameters.StartDirection 		:= mcDIR_POSITIVE;
	//			fbMovelVel.AdvancedParameters.EndDirection 			:= mcDIR_UNDEFINED;
	//			fbMovelVel.AdvancedParameters.ShuttleOrientation 	:= mcDIR_UNDEFINED;
	//
	//			IF bMoveVelActive = FALSE AND fbMovelVel.Active = TRUE THEN
	//				fbMovelVel.Execute 		:= FALSE;
	//				initStep 				:= 122;
	//			END_IF
	//
	//		122:
	//			IF fbSecGetShuttles.RemainingCount > 0 THEN
	//				fbSecGetShuttles.Next 		:= TRUE;
	//				initStep 				:= 121;
	//			ELSE
	//				fbSecGetShuttles.Enable := FALSE;
	//				initStep 				:= 130;
	//			END_IF
	//			////////////////////////////////////////////////////////////////////////
	//		130:
	//			fbSecGetShuttles.Sector := ADR(SecMain);
	//			fbSecGetShuttles.Enable := TRUE;
	//			fbSecGetShuttles.AdvancedParameters.StartPosition := 0.0;
	//			fbSecGetShuttles.AdvancedParameters.EndPosition := 0.0;
	//
	//			IF fbSecGetShuttles.Valid = TRUE THEN
	//				IF fbSecGetShuttles.TotalCount > 0 THEN
	//					initStep 					:= 131;
	//				ELSE
	//					fbSecGetShuttles.Enable 	:= FALSE;
	//					initStep 					:= 140;
	//				END_IF
	//			END_IF
	//
	//		131:
	//			fbSecGetShuttles.Next 			:= FALSE;
	//
	//			fbMovelVel.Sector				:= ADR(SecMain);
	//			fbMovelVel.Axis 				:= ADR(fbSecGetShuttles.Axis);
	//
	//			fbMovelVel.RouteVelocity 		:= gPar.MovementPar.Initialize.RoutedVelocity;
	//			fbMovelVel.Velocity 			:= gPar.MovementPar.Initialize.Velocity;
	//			fbMovelVel.Acceleration 		:= gPar.MovementPar.Initialize.Acceleration;
	//			fbMovelVel.Deceleration 		:= gPar.MovementPar.Initialize.Deceleration;
	//			fbMovelVel.Execute 				:= TRUE;
	//
	//			fbMovelVel.AdvancedParameters.StartDirection 		:= mcDIR_POSITIVE;
	//			fbMovelVel.AdvancedParameters.EndDirection 			:= mcDIR_UNDEFINED;
	//			fbMovelVel.AdvancedParameters.ShuttleOrientation 	:= mcDIR_UNDEFINED;
	//
	//			IF bMoveVelActive = FALSE AND fbMovelVel.Active = TRUE THEN
	//				fbMovelVel.Execute 			:= FALSE;
	//				initStep 					:= 132;
	//			END_IF
	//
	//		132:
	//			IF fbSecGetShuttles.RemainingCount > 0 THEN
	//				fbSecGetShuttles.Next 		:= TRUE;
	//				initStep 					:= 131;
	//			ELSE
	//				fbSecGetShuttles.Enable 	:= FALSE;
	//				initStep 					:= 140;
	//			END_IF
	//			////////////////////////////////////////////////////////////////////////
	//		140:
	//			fbSecGetShuttles.Sector := ADR(SecIn);
	//			fbSecGetShuttles.Enable := TRUE;
	//			fbSecGetShuttles.AdvancedParameters.StartPosition := 2.55;
	//			fbSecGetShuttles.AdvancedParameters.EndPosition := 0.0;
	//
	//			IF fbSecGetShuttles.Valid = TRUE THEN
	//				IF fbSecGetShuttles.TotalCount > 0 THEN
	//					initStep 					:= 141;
	//				ELSE
	//					fbSecGetShuttles.Enable 	:= FALSE;
	//					initStep 					:= 150;
	//				END_IF
	//			END_IF
	//
	//		141:
	//			fbSecGetShuttles.Next 			:= FALSE;
	//
	//			fbMovelVel.Sector				:= ADR(SecMain);
	//			fbMovelVel.Axis 				:= ADR(fbSecGetShuttles.Axis);
	//
	//			fbMovelVel.RouteVelocity 		:= gPar.MovementPar.Initialize.RoutedVelocity;
	//			fbMovelVel.Velocity 			:= gPar.MovementPar.Initialize.Velocity;
	//			fbMovelVel.Acceleration 		:= gPar.MovementPar.Initialize.Acceleration;
	//			fbMovelVel.Deceleration 		:= gPar.MovementPar.Initialize.Deceleration;
	//			fbMovelVel.Execute 				:= TRUE;
	//
	//			fbMovelVel.AdvancedParameters.StartDirection 		:= mcDIR_NEGATIVE;
	//			fbMovelVel.AdvancedParameters.EndDirection 			:= mcDIR_UNDEFINED;
	//			fbMovelVel.AdvancedParameters.ShuttleOrientation 	:= mcDIR_UNDEFINED;
	//
	//			IF bMoveVelActive = FALSE AND fbMovelVel.Active = TRUE THEN
	//				fbMovelVel.Execute 			:= FALSE;
	//				initStep 					:= 142;
	//			END_IF
	//
	//		142:
	//			IF fbSecGetShuttles.RemainingCount > 0 THEN
	//				fbSecGetShuttles.Next 		:= TRUE;
	//				initStep 					:= 141;
	//			ELSE
	//				fbSecGetShuttles.Enable 	:= FALSE;
	//				initStep 					:= 150;
	//			END_IF
	//			////////////////////////////////////////////////////////////////////////
	//		150:
	//			fbSecGetShuttles.Sector := ADR(SecOut);
	//			fbSecGetShuttles.Enable := TRUE;
	//			fbSecGetShuttles.AdvancedParameters.StartPosition := 0.0;
	//			fbSecGetShuttles.AdvancedParameters.EndPosition := 1.13;
	//
	//			IF fbSecGetShuttles.Valid = TRUE THEN
	//				IF fbSecGetShuttles.TotalCount > 0 THEN
	//					fbSecGetShuttles.Enable 	:= FALSE;
	//					initStep 					:= 150;
	//				ELSE
	//					fbSecGetShuttles.Enable 	:= FALSE;
	//					initStep 					:= 160;
	//				END_IF
	//			END_IF
	//			////////////////////////////////////////////////////////////////////////
	//		160:
	//			fbSecGetShuttles.Sector := ADR(SecIn);
	//			fbSecGetShuttles.Enable := TRUE;
	//			fbSecGetShuttles.AdvancedParameters.StartPosition := 0.0;
	//			fbSecGetShuttles.AdvancedParameters.EndPosition := 0.0;
	//
	//			IF fbSecGetShuttles.Valid = TRUE THEN
	//				IF fbSecGetShuttles.TotalCount > 0 THEN
	//					initStep 					:= 161;
	//				ELSE
	//					fbSecGetShuttles.Enable 	:= FALSE;
	//					initStep 					:= 170;
	//				END_IF
	//			END_IF
	//
	//		161:
	//			fbSecGetShuttles.Next 			:= FALSE;
	//
	//			fbMovelVel.Sector				:= ADR(SecMain);
	//			fbMovelVel.Axis 				:= ADR(fbSecGetShuttles.Axis);
	//
	//			fbMovelVel.RouteVelocity 		:= gPar.MovementPar.Initialize.RoutedVelocity;
	//			fbMovelVel.Velocity 			:= gPar.MovementPar.Initialize.Velocity;
	//			fbMovelVel.Acceleration 		:= gPar.MovementPar.Initialize.Acceleration;
	//			fbMovelVel.Deceleration 		:= gPar.MovementPar.Initialize.Deceleration;
	//			fbMovelVel.Execute 				:= TRUE;
	//
	//			fbMovelVel.AdvancedParameters.StartDirection 		:= mcDIR_NEGATIVE;
	//			fbMovelVel.AdvancedParameters.EndDirection 			:= mcDIR_POSITIVE;
	//			fbMovelVel.AdvancedParameters.ShuttleOrientation 	:= mcDIR_UNDEFINED;
	//
	//			IF bMoveVelActive = FALSE AND fbMovelVel.Active = TRUE THEN
	//				fbMovelVel.Execute 			:= FALSE;
	//				initStep 					:= 162;
	//			END_IF
	//
	//		162:
	//			IF fbSecGetShuttles.RemainingCount > 0 THEN
	//				fbSecGetShuttles.Next 		:= TRUE;
	//				initStep 					:= 161;
	//			ELSE
	//				fbSecGetShuttles.Enable 	:= FALSE;
	//				initStep 					:= 170;
	//			END_IF
	//
	//		170:
	//			fbBarGetShuttle.ProcessPoint 	:= ADR(ptBufferIn);
	////			fbBarGetShuttle.Enable 			:= TRUE;
	//			fbBarGetShuttle;
	//
	//		200:
	//			fbBarBufferOut.Command			:= mcACPTRAK_BARRIER_OPEN;
	//			fbBarBufferOut.Execute 			:= TRUE;
	//
	//			fbBarCmd.Command 				:= mcACPTRAK_BARRIER_OPEN;
	//			fbBarCmd.Execute 				:= TRUE;
	//
	//			IF fbBarCmd.Done = TRUE AND fbBarBufferOut.Done = TRUE THEN
	//				fbBarBufferOut.Execute 		:= FALSE;
	//				fbBarCmd.Execute 			:= FALSE;
	//				initStep 					:= 300;
	//			END_IF
	//
	//		300:
	//			gSts.AsmState 					:= E_ASM_IDLE;
	//			initStep 						:= 0;
	//
	//	END_CASE;

	//	fbBarNG();
	//	fbBarCmd();
	//	fbBarBufferOut();
	//	fbSecGetShuttles();
	//
	//	bMoveVelActive := fbMovelVel.Active;
	//
	//	fbMovelVel();
END_PROGRAM
```

### Program Logical/Source/AsmControl/ctrMaint (IEC) - Maint Control

#### Types.typ
```iecst
TYPE
	E_MAINT_STEP :
		(
		E_MAINT_DIABLE := 0,
		E_MAINT_LINK_CURRENT_SH := 100,
		E_MAINT_SELECTED_SHUTTLE := 200,
		E_MAINT_RUN_ABS := 300,
		E_MAINT_RUN_VEL := 400
		);
END_TYPE
```

#### Variables.var
```iecst
VAR
	fbAsmGetShuttle : MC_BR_AsmGetShuttle_AcpTrak;
	fbRoutedMoveAbs : MC_BR_RoutedMoveAbs_AcpTrak;
	fbReadShuttleInfo : MC_BR_ShReadInfo_AcpTrak;
	fbStop : MC_Stop;
	fbGetUserData : MC_BR_ShCopyUserData_AcpTrak;
END_VAR
(**)
VAR
	cmdNextSh : R_TRIG;
	cmdMoveAbs : R_TRIG;
	cmdStop : R_TRIG;
END_VAR
(**)
VAR
	Step : E_MAINT_STEP; (*Step*)
	UserData : ShuttleUserData_typ; (*User Data of Selected Shuttle*)
	NextShuttle : BOOL; (*Connect to Next Shuttle*)
	MaintShuttleControlEnable : BOOL; (*Maint Controller Enable*)
	CurrentShuttleIndex : UINT; (*Current Shuttle Index*)
	MoveAbsolute : BOOL; (*Maint Controller Enable*)
	Stop : BOOL; (*Maint Controller Enable*)
END_VAR
```

#### Main.st
```iecst
PROGRAM _INIT
	fbAsmGetShuttle.Assembly 	:= ADR(gAsmMain);

	fbRoutedMoveAbs.Sector := ADR(SectorTrackAll);

	fbGetUserData.Axis			:= ADR(fbAsmGetShuttle.Axis);
	fbReadShuttleInfo.Axis 		:= ADR(fbAsmGetShuttle.Axis);
	fbStop.Axis					:= ADR(fbAsmGetShuttle.Axis);
	fbRoutedMoveAbs.Axis 		:= ADR(fbAsmGetShuttle.Axis);

	fbGetUserData.DataAddress	:= ADR(UserData);
	fbGetUserData.DataSize		:= SIZEOF(UserData);
END_PROGRAM

PROGRAM _CYCLIC
	IF fbAsmGetShuttle.Error = TRUE THEN
		MaintShuttleControlEnable 	:= FALSE;
		Step 						:= E_MAINT_DIABLE;
	END_IF

	cmdStop(CLK := Stop);
	cmdNextSh(CLK := NextShuttle);
	cmdMoveAbs(CLK := MoveAbsolute);

	IF cmdStop.Q = TRUE THEN
		fbStop.Execute := TRUE;
	END_IF

	CASE Step OF
		E_MAINT_DIABLE:
			IF gSts.AsmState = E_ASM_ON AND MaintShuttleControlEnable = TRUE THEN
				fbAsmGetShuttle.Enable 	:= TRUE;

				IF fbAsmGetShuttle.Valid = TRUE THEN
					CurrentShuttleIndex := fbAsmGetShuttle.RemainingCount + 1;
					Step 				:= E_MAINT_LINK_CURRENT_SH;
				END_IF
			ELSE
				fbAsmGetShuttle.Enable 	:= FALSE;
			END_IF

		E_MAINT_LINK_CURRENT_SH:
			fbReadShuttleInfo.Enable 		:= TRUE;
			fbGetUserData.Execute 			:= TRUE;

			fbAsmGetShuttle.Next 			:= FALSE;

			IF fbGetUserData.Done = TRUE AND fbReadShuttleInfo.Valid = TRUE THEN
				fbGetUserData.Execute		:= FALSE;
				Step 						:= E_MAINT_SELECTED_SHUTTLE;
			END_IF

		E_MAINT_SELECTED_SHUTTLE:
			IF cmdNextSh.Q = TRUE THEN
				fbReadShuttleInfo.Enable 		:= FALSE;

				IF fbAsmGetShuttle.RemainingCount > 0 THEN
					fbAsmGetShuttle.Next 	:= TRUE;
					Step 					:= E_MAINT_LINK_CURRENT_SH;
				ELSE
					fbAsmGetShuttle.Enable := FALSE;
					Step 					:= E_MAINT_DIABLE;
				END_IF
			ELSIF cmdMoveAbs.Q = TRUE THEN
				Step 						:= E_MAINT_RUN_ABS;
			END_IF

		E_MAINT_RUN_ABS:
			fbRoutedMoveAbs.Execute 	:= TRUE;

			IF fbRoutedMoveAbs.Done = TRUE OR fbRoutedMoveAbs.CommandAborted = TRUE OR fbRoutedMoveAbs.Error = TRUE THEN
				Step 						:= E_MAINT_SELECTED_SHUTTLE;
				fbRoutedMoveAbs.Execute 	:= FALSE;

			END_IF
	END_CASE

	IF fbStop.Error = TRUE OR fbStop.Done = TRUE THEN
		fbStop.Execute := FALSE;
	END_IF

	MoveAbsolute				:= FALSE;
	Stop						:= FALSE;

	fbStop;
	fbGetUserData;
	fbRoutedMoveAbs;
	fbAsmGetShuttle;
	fbReadShuttleInfo;
END_PROGRAM
```

### Program Logical/Source/AsmControl/ctrTeaching (IEC) - Teaching in Manual Mode

#### Types.typ
```iecst
TYPE
	E_STAGE_LIST :
		(
		E_STAGE_NONE := 0,
		E_STAGE_STAGE1 := 1,
		E_STAGE_STAGE2 := 2,
		E_STAGE_STAGE3 := 3,
		E_STAGE_STAGE4 := 4,
		E_STAGE_STAGE5 := 5,
		E_STAGE_STAGE6 := 6,
		E_STAGE_STAGE7 := 7,
		E_STAGE_STAGE8 := 8,
		E_STAGE_STAGE9 := 9,
		E_STAGE_STAGE10 := 10,
		E_STAGE_STAGE11 := 11,
		E_STAGE_STAGE12 := 12,
		E_STAGE_STAGE13 := 13,
		E_STAGE_STAGE14 := 14,
		E_STAGE_STAGE15 := 15,
		E_STAGE_STAGE16 := 16,
		E_STAGE_STAGE17 := 17,
		E_STAGE_STAGE18 := 18,
		E_STAGE_STAGE19 := 19
		);
END_TYPE
```

#### Variables.var
```iecst
VAR
	step : UDINT;
	selectedStage : E_STAGE_LIST;
	openDialog : BOOL;
	execute : BOOL;
	apply : BOOL;
	position : LREAL;
	position_max : LREAL;
	position_min : LREAL;
END_VAR
(**)
VAR
	r_trgExecute : R_TRIG;
	r_trgApply : R_TRIG;
	elasticAbsMove : MC_BR_ElasticMoveAbs_AcpTrak;
END_VAR
```

#### Main.st
```iecst
PROGRAM _INIT
	elasticAbsMove.Velocity 		:= 0.5;
	elasticAbsMove.Acceleration 	:= 1.0;
	elasticAbsMove.Deceleration 	:= 1.0;

END_PROGRAM

PROGRAM _CYCLIC
	r_trgExecute(CLK := execute);
	r_trgApply(CLK := apply);

	CASE step OF
		0:	(*Manual IDLE*)
			IF selectedStage <> E_STAGE_NONE THEN
				IF selectedStage = E_STAGE_STAGE1 AND StStage[0].Shuttle.controlif <> 0 THEN
					elasticAbsMove.Axis 	:= ADR(StStage[0].Shuttle);
					position				:= (gPar.ProcessPosition.Stage[0]);
					position_max			:= POS_STAGE1_MAX;
					position_min			:= POS_STAGE1_MIN;
				ELSIF selectedStage = E_STAGE_STAGE2	AND StStage[1].Shuttle.controlif <> 0 THEN
					elasticAbsMove.Axis 	:= ADR(StStage[1].Shuttle);
					position				:= (gPar.ProcessPosition.Stage[1]);
					position_max			:= POS_STAGE2_MAX;
					position_min			:= POS_STAGE2_MAX;
				ELSIF selectedStage = E_STAGE_STAGE3	AND StStage[2].Shuttle.controlif <> 0 THEN
					elasticAbsMove.Axis 	:= ADR(StStage[2].Shuttle);
					position				:= (gPar.ProcessPosition.Stage[2]);
					position_max			:= POS_STAGE3_MAX;
					position_min			:= POS_STAGE3_MAX;
				ELSIF selectedStage = E_STAGE_STAGE4	AND StStage[3].Shuttle.controlif <> 0 THEN
					elasticAbsMove.Axis 	:= ADR(StStage[3].Shuttle);
					position				:= (gPar.ProcessPosition.Stage[3]);
					position_max			:= POS_STAGE4_MAX;
					position_min			:= POS_STAGE4_MAX;
				ELSIF selectedStage = E_STAGE_STAGE5	AND StStage[4].Shuttle.controlif <> 0 THEN
					elasticAbsMove.Axis 	:= ADR(StStage[4].Shuttle);
					position				:= (gPar.ProcessPosition.Stage[4]);
					position_max			:= POS_STAGE5_MAX;
					position_min			:= POS_STAGE5_MAX;
				ELSIF selectedStage = E_STAGE_STAGE6	AND StStage[5].Shuttle.controlif <> 0 THEN
					elasticAbsMove.Axis 	:= ADR(StStage[5].Shuttle);
					position				:= (gPar.ProcessPosition.Stage[5]);
					position_max			:= POS_STAGE6_MAX;
					position_min			:= POS_STAGE6_MAX;
				ELSIF selectedStage = E_STAGE_STAGE7	AND StStage[6].Shuttle.controlif <> 0 THEN
					elasticAbsMove.Axis 	:= ADR(StStage[6].Shuttle);
					position				:= (gPar.ProcessPosition.Stage[6]);
					position_max			:= POS_STAGE7_MAX;
					position_min			:= POS_STAGE7_MAX;
				ELSIF selectedStage = E_STAGE_STAGE8	AND StStage[7].Shuttle.controlif <> 0 THEN
					elasticAbsMove.Axis 	:= ADR(StStage[7].Shuttle);
					position				:= (gPar.ProcessPosition.Stage[7]);
					position_max			:= POS_STAGE8_MAX;
					position_min			:= POS_STAGE8_MAX;
				ELSIF selectedStage = E_STAGE_STAGE9	AND StStage[8].Shuttle.controlif <> 0 THEN
					elasticAbsMove.Axis 	:= ADR(StStage[8].Shuttle);
					position				:= (gPar.ProcessPosition.Stage[8]);
					position_max			:= POS_STAGE9_MAX;
					position_min			:= POS_STAGE9_MAX;
				ELSIF selectedStage = E_STAGE_STAGE10	AND StStage[9].Shuttle.controlif <> 0 THEN
					elasticAbsMove.Axis 	:= ADR(StStage[9].Shuttle);
					position				:= (gPar.ProcessPosition.Stage[9]);
					position_max			:= POS_STAGE10_MAX;
					position_min			:= POS_STAGE10_MAX;
				ELSIF selectedStage = E_STAGE_STAGE11	AND StStage[10].Shuttle.controlif <> 0 THEN
					elasticAbsMove.Axis 	:= ADR(StStage[10].Shuttle);
					position				:= (gPar.ProcessPosition.Stage[10]);
					position_max			:= POS_STAGE11_MAX;
					position_min			:= POS_STAGE11_MAX;
				ELSIF selectedStage = E_STAGE_STAGE12	AND StStage[11].Shuttle.controlif <> 0 THEN
					elasticAbsMove.Axis 	:= ADR(StStage[11].Shuttle);
					position				:= (gPar.ProcessPosition.Stage[11]);
					position_max			:= POS_STAGE12_MAX;
					position_min			:= POS_STAGE12_MAX;
				ELSIF selectedStage = E_STAGE_STAGE13	AND StStage[12].Shuttle.controlif <> 0 THEN
					elasticAbsMove.Axis 	:= ADR(StStage[12].Shuttle);
					position				:= (gPar.ProcessPosition.Stage[12]);
					position_max			:= POS_STAGE13_MAX;
					position_min			:= POS_STAGE13_MAX;
				ELSIF selectedStage = E_STAGE_STAGE14	AND StStage[13].Shuttle.controlif <> 0 THEN
					elasticAbsMove.Axis 	:= ADR(StStage[13].Shuttle);
					position				:= (gPar.ProcessPosition.Stage[13]);
					position_max			:= POS_STAGE14_MAX;
					position_min			:= POS_STAGE14_MAX;
				ELSIF selectedStage = E_STAGE_STAGE15	AND StStage[14].Shuttle.controlif <> 0 THEN
					elasticAbsMove.Axis 	:= ADR(StStage[14].Shuttle);
					position				:= (gPar.ProcessPosition.Stage[14]);
					position_max			:= POS_STAGE15_MAX;
					position_min			:= POS_STAGE15_MAX;
				ELSIF selectedStage = E_STAGE_STAGE16	AND StStage[15].Shuttle.controlif <> 0 THEN
					elasticAbsMove.Axis 	:= ADR(StStage[15].Shuttle);
					position				:= (gPar.ProcessPosition.Stage[15]);
					position_max			:= POS_STAGE16_MAX;
					position_min			:= POS_STAGE16_MAX;
				ELSIF selectedStage = E_STAGE_STAGE17	AND StStage[16].Shuttle.controlif <> 0 THEN
					elasticAbsMove.Axis 	:= ADR(StStage[16].Shuttle);
					position				:= (gPar.ProcessPosition.Stage[16]);
					position_max			:= POS_STAGE17_MAX;
					position_min			:= POS_STAGE17_MAX;
				ELSIF selectedStage = E_STAGE_STAGE18	AND StStage[17].Shuttle.controlif <> 0 THEN
					elasticAbsMove.Axis 	:= ADR(StStage[17].Shuttle);
					position				:= (gPar.ProcessPosition.Stage[17]);
					position_max			:= POS_STAGE18_MAX;
					position_min			:= POS_STAGE18_MAX;
				ELSIF selectedStage = E_STAGE_STAGE19	AND StStage[18].Shuttle.controlif <> 0 THEN
					elasticAbsMove.Axis 	:= ADR(StStage[18].Shuttle);
					position				:= (gPar.ProcessPosition.Stage[18]);
					position_max			:= POS_STAGE19_MAX;
					position_min			:= POS_STAGE19_MAX;
				END_IF

				openDialog				:= TRUE;
				step 					:= 100;
			END_IF

		100: (*Manual RUN*)
			IF r_trgExecute.Q = TRUE THEN
				elasticAbsMove.Position := position;
				elasticAbsMove.Execute	:= TRUE;
				step 					:= 110;
			ELSIF r_trgApply.Q = TRUE THEN
				IF selectedStage = E_STAGE_STAGE1 THEN
					gPar.ProcessPosition.Stage[0] := position;
				ELSIF selectedStage = E_STAGE_STAGE2 THEN
					gPar.ProcessPosition.Stage[1] := position;
				ELSIF selectedStage = E_STAGE_STAGE3 THEN
					gPar.ProcessPosition.Stage[2] := position;
				ELSIF selectedStage = E_STAGE_STAGE4 THEN
					gPar.ProcessPosition.Stage[3] := position;
				ELSIF selectedStage = E_STAGE_STAGE5 THEN
					gPar.ProcessPosition.Stage[4] := position;
				ELSIF selectedStage = E_STAGE_STAGE6 THEN
					gPar.ProcessPosition.Stage[5] := position;
				ELSIF selectedStage = E_STAGE_STAGE7 THEN
					gPar.ProcessPosition.Stage[6] := position;
				ELSIF selectedStage = E_STAGE_STAGE8 THEN
					gPar.ProcessPosition.Stage[7] := position;
				ELSIF selectedStage = E_STAGE_STAGE9 THEN
					gPar.ProcessPosition.Stage[8] := position;
				ELSIF selectedStage = E_STAGE_STAGE10 THEN
					gPar.ProcessPosition.Stage[9] := position;
				ELSIF selectedStage = E_STAGE_STAGE11 THEN
					gPar.ProcessPosition.Stage[10] := position;
				ELSIF selectedStage = E_STAGE_STAGE12 THEN
					gPar.ProcessPosition.Stage[11] := position;
				ELSIF selectedStage = E_STAGE_STAGE13 THEN
					gPar.ProcessPosition.Stage[12] := position;
				ELSIF selectedStage = E_STAGE_STAGE14 THEN
					gPar.ProcessPosition.Stage[13] := position;
				ELSIF selectedStage = E_STAGE_STAGE15 THEN
					gPar.ProcessPosition.Stage[14] := position;
				ELSIF selectedStage = E_STAGE_STAGE16 THEN
					gPar.ProcessPosition.Stage[15] := position;
				ELSIF selectedStage = E_STAGE_STAGE17 THEN
					gPar.ProcessPosition.Stage[16] := position;
				ELSIF selectedStage = E_STAGE_STAGE18 THEN
					gPar.ProcessPosition.Stage[17] := position;
				ELSIF selectedStage = E_STAGE_STAGE19 THEN
					gPar.ProcessPosition.Stage[18] := position;
				END_IF

				elasticAbsMove.Axis 	:= 0;
				step 					:= 0;
				openDialog				:= FALSE;
				elasticAbsMove.Execute 	:= FALSE;
				selectedStage 			:= E_STAGE_NONE;
			ELSIF selectedStage = E_STAGE_NONE THEN
				elasticAbsMove.Axis 	:= 0;
				step 					:= 0;
				openDialog				:= FALSE;
				elasticAbsMove.Execute 	:= FALSE;
			END_IF

		110:
			IF elasticAbsMove.Done = TRUE THEN
				elasticAbsMove.Execute	:= FALSE;
				step := 100;
			ELSIF elasticAbsMove.Error = TRUE THEN
				elasticAbsMove.Execute	:= FALSE;
				step := 100;
			END_IF

	END_CASE;

	elasticAbsMove();

	execute 	:= FALSE;
	apply 		:= FALSE;
END_PROGRAM

PROGRAM _EXIT
	(* Insert code here *)

END_PROGRAM
```

### Program Logical/Source/AsmControl/ctrCodeReader (IEC)

#### Main.st - Init, cyclic, exit code
```iecst
PROGRAM _INIT
	(* Insert code here *)

	fbTrig.ProcessPoint			:= ADR(ptVision);
	fbTrigInfo.ProcessPoint		:= ADR(ptVision);

	ShReadInfo.Axis 	:= ADR(Axis);

	fbUserData.Axis	:= ADR(fbTrigInfo.TrgPointInfo);

	fbTrig();
	fbTrigInfo();
	fbUserData();
	ShReadInfo();

END_PROGRAM

PROGRAM _CYCLIC
	(* Insert code here *)

	gBarCodeReader.Enable 		:= TRUE;

	CASE gSts.AsmState OF

		E_ASM_INITIALIZATION:

			IF NOT gSim THEN
				gInitialDone		:= FALSE;
			END_IF

			actCodeReader;

		E_ASM_IDLE:

			actCodeReader;

		ELSE
			actCodeReader_INIT;

	END_CASE

	fbTrig();
	fbTrigInfo();
	fbUserData();
	ShReadInfo();

END_PROGRAM

PROGRAM _EXIT
	(* Insert code here *)

END_PROGRAM
```

#### Types.typ - Local data types
```iecst
TYPE
	E_CODE_STEP :
		(
		CODE_WAIT := 0,
		CODE_CHECK_TRIG := 100,
		CODE_GET_SH := 200,
		CODE_MOVE_TO_READER := 300,
		CODE_READER_CHECK := 400,
		CODE_CHECK_TAKE_COUNT := 500,
		CODE_ID_DEFINE := 600,
		CODE_RELEASE_SH := 700,
		CODE_NORMAL_END := 1000
		) := CODE_WAIT;
END_TYPE
```

#### Variables.var - Local variables
```iecst
VAR
	CodeStep : E_CODE_STEP;
END_VAR
(**)
VAR
	fbMovelVel : MC_BR_RoutedMoveVel_AcpTrak;
	fbMovelAbs : MC_BR_RoutedMoveAbs_AcpTrak;
	fbTrigInfo : MC_BR_TrgPointGetInfo_AcpTrak;
	fbTrig : MC_BR_TrgPointEnable_AcpTrak;
	ShReadInfo : MC_BR_ShReadInfo_AcpTrak;
	Axis : McAxisType;
	userData : ShuttleUserData_typ;
	fbUserData : MC_BR_ShCopyUserData_AcpTrak;
	checkTakeCount : USINT;
	checkSHCount : USINT;
	bMoveVelActive : BOOL;
	StrShuttleCount : STRING[80];
	StrTempShuttleID : STRING[80];
	bNextStep1 : BOOL;
	bNextStep2 : BOOL;
	bNextStep3 : BOOL;
	bNextStep4 : BOOL;
END_VAR
```
